//-------------------------------------------------------------------------------------------------------------------
//-- Stop --
	//
	TPL.FC_FirstStep(udiStepIndex, diStep);
	astStopTable[udiStepIndex].sTitle						:= 'Stop AllSubModules';
	astStopTable[udiStepIndex].udiModuleName				:= TPL.Gc_udiAllSubModules;
	astStopTable[udiStepIndex].diStep						:= diStep;
	astStopTable[udiStepIndex].diCMD						:= AXM.ET_Cmd.Stop;
	astStopTable[udiStepIndex].timTimeOut					:= T#0MS;
	astStopTable[udiStepIndex].xEndCMD						:= FALSE;
	
	TPL.FC_LastStep(udiStepIndex, diStep);
	astStopTable[udiStepIndex].sTitle						:= 'End';
	astStopTable[udiStepIndex].udiModuleName				:= 0;
	astStopTable[udiStepIndex].diStep						:= diStep;
	astStopTable[udiStepIndex].diCMD						:= 0;
	astStopTable[udiStepIndex].timTimeOut					:= T#0MS;
	astStopTable[udiStepIndex].xEndCMD						:= TRUE;
	
	TPL.FC_NextCmdTable(iq_udiTableIndex:= udiTableIndex);
	astListofCMDTables[udiTableIndex].sTitle				:= 'Stop';
	astListofCMDTables[udiTableIndex].diCMD					:= ET_Cmd.Stop;
	astListofCMDTables[udiTableIndex].udiNumberOfCmdSteps	:= udiStepIndex;

//-------------------------------------------------------------------------------------------------------------------
//-- Start --
	//
	TPL.FC_FirstStep(udiStepIndex, diStep);
	astStartTable[udiStepIndex].sTitle						:= 'Start AllSubModules';
	astStartTable[udiStepIndex].udiModuleName				:= TPL.Gc_udiAllSubModules;
	astStartTable[udiStepIndex].diStep						:= diStep;
	astStartTable[udiStepIndex].diCMD						:= AXM.ET_Cmd.Start;
	astStartTable[udiStepIndex].timTimeOut					:= T#0MS;
	astStartTable[udiStepIndex].xEndCMD						:= FALSE;
	
	TPL.FC_LastStep(udiStepIndex, diStep);
	astStartTable[udiStepIndex].sTitle						:= 'End';
	astStartTable[udiStepIndex].udiModuleName				:= 0;
	astStartTable[udiStepIndex].diStep						:= diStep;
	astStartTable[udiStepIndex].diCMD						:= 0;
	astStartTable[udiStepIndex].timTimeOut					:= T#0MS;
	astStartTable[udiStepIndex].xEndCMD						:= TRUE;
	
	TPL.FC_NextCmdTable(iq_udiTableIndex:= udiTableIndex);
	astListofCMDTables[udiTableIndex].sTitle				:= 'Start';
	astListofCMDTables[udiTableIndex].diCMD					:= ET_Cmd.Start;
	astListofCMDTables[udiTableIndex].udiNumberOfCmdSteps	:= udiStepIndex;
	
//-------------------------------------------------------------------------------------------------------------------
//-- Abort --
	//
	TPL.FC_FirstStep(udiStepIndex, diStep);
	astAbortTable[udiStepIndex].sTitle						:= 'Stop AllSubModules';
	astAbortTable[udiStepIndex].udiModuleName				:= TPL.Gc_udiAllSubModules;
	astAbortTable[udiStepIndex].diStep						:= diStep;
	astAbortTable[udiStepIndex].diCMD						:= AXM.ET_Cmd.Stop;
	astAbortTable[udiStepIndex].timTimeOut					:= T#0MS;
	astAbortTable[udiStepIndex].xEndCMD						:= FALSE;
	
	TPL.FC_LastStep(udiStepIndex, diStep);
	astAbortTable[udiStepIndex].sTitle						:= 	'End';
	astAbortTable[udiStepIndex].udiModuleName				:= 	0;
	astAbortTable[udiStepIndex].diStep						:= 	diStep;
	astAbortTable[udiStepIndex].diCMD						:= 	0;
	astAbortTable[udiStepIndex].timTimeOut					:=	T#0MS;
	astAbortTable[udiStepIndex].xEndCMD						:= TRUE;
	
	TPL.FC_NextCmdTable(iq_udiTableIndex:= udiTableIndex);
	astListofCMDTables[udiTableIndex].sTitle				:= 'Abort';
	astListofCMDTables[udiTableIndex].diCMD					:= ET_Cmd.Abort;
	astListofCMDTables[udiTableIndex].udiNumberOfCmdSteps	:= udiStepIndex;

//-------------------------------------------------------------------------------------------------------------------
//-- Hold --
	//
	TPL.FC_FirstStep(udiStepIndex, diStep);
	astHoldTable[udiStepIndex].sTitle						:= 'Hold AllSubModules';
	astHoldTable[udiStepIndex].udiModuleName				:= TPL.Gc_udiAllSubModules;
	astHoldTable[udiStepIndex].diStep						:= diStep;
	astHoldTable[udiStepIndex].diCMD						:= AXM.ET_Cmd.Hold;
	astHoldTable[udiStepIndex].timTimeOut					:= T#0MS;
	astHoldTable[udiStepIndex].xEndCMD						:= FALSE;
	
	TPL.FC_LastStep(udiStepIndex, diStep);
	astHoldTable[udiStepIndex].sTitle						:= 'End';
	astHoldTable[udiStepIndex].udiModuleName				:= 0;
	astHoldTable[udiStepIndex].diStep						:= diStep;
	astHoldTable[udiStepIndex].diCMD						:= 0;
	astHoldTable[udiStepIndex].timTimeOut					:= T#0MS;
	astHoldTable[udiStepIndex].xEndCMD						:= TRUE;
	
	TPL.FC_NextCmdTable(iq_udiTableIndex:= udiTableIndex);
	astListofCMDTables[udiTableIndex].sTitle				:= 'Hold';
	astListofCMDTables[udiTableIndex].diCMD					:= ET_Cmd.Hold;
	astListofCMDTables[udiTableIndex].udiNumberOfCmdSteps	:= udiStepIndex;

//-------------------------------------------------------------------------------------------------------------------
//-- Brake Release --
	//
	TPL.FC_FirstStep(udiStepIndex, diStep);
	astBrakeReleaseTable[udiStepIndex].sTitle				:= 'AxisEnable Off AllSubModules';
	astBrakeReleaseTable[udiStepIndex].udiModuleName		:= TPL.Gc_udiAllSubModules;
	astBrakeReleaseTable[udiStepIndex].diStep				:= diStep;
	astBrakeReleaseTable[udiStepIndex].diCMD				:= AXM.ET_Cmd.DriveEnableOff;
	astBrakeReleaseTable[udiStepIndex].timTimeOut			:= T#0MS;
	astBrakeReleaseTable[udiStepIndex].xEndCMD				:= FALSE;
	
	TPL.FC_NextStep(udiStepIndex, diStep);
	astBrakeReleaseTable[udiStepIndex].sTitle				:= 'BrakeRelease Mode AllSubModules';
	astBrakeReleaseTable[udiStepIndex].udiModuleName		:= TPL.Gc_udiAllSubModules;
	astBrakeReleaseTable[udiStepIndex].diStep				:= diStep;
	astBrakeReleaseTable[udiStepIndex].diCMD				:= AXM.ET_Cmd.BrakeRelease;
	astBrakeReleaseTable[udiStepIndex].timTimeOut			:= T#0MS;
	astBrakeReleaseTable[udiStepIndex].xEndCMD				:= FALSE;
	
	TPL.FC_NextStep(udiStepIndex, diStep);
	astBrakeReleaseTable[udiStepIndex].sTitle				:= 'Start AllSubModules';
	astBrakeReleaseTable[udiStepIndex].udiModuleName		:= TPL.Gc_udiAllSubModules;
	astBrakeReleaseTable[udiStepIndex].diStep				:= diStep;
	astBrakeReleaseTable[udiStepIndex].diCMD				:= AXM.ET_Cmd.Start;
	astBrakeReleaseTable[udiStepIndex].timTimeOut			:= T#0MS;
	astBrakeReleaseTable[udiStepIndex].xEndCMD				:= FALSE;
	
	TPL.FC_LastStep(udiStepIndex, diStep);
	astBrakeReleaseTable[udiStepIndex].sTitle				:= 'End';
	astBrakeReleaseTable[udiStepIndex].udiModuleName		:= 0;
	astBrakeReleaseTable[udiStepIndex].diStep				:= diStep;
	astBrakeReleaseTable[udiStepIndex].diCMD				:= 0;
	astBrakeReleaseTable[udiStepIndex].timTimeOut			:= T#0MS;
	astBrakeReleaseTable[udiStepIndex].xEndCMD				:= TRUE;
	
	TPL.FC_NextCmdTable(iq_udiTableIndex:= udiTableIndex);
	astListofCMDTables[udiTableIndex].sTitle				:= 'Brake Release';
	astListofCMDTables[udiTableIndex].diCMD					:= ET_Cmd.BrakeRelease;
	astListofCMDTables[udiTableIndex].udiNumberOfCmdSteps	:= udiStepIndex;
	//
//
			
// End of system generated code, could be modified for your application -)
END_ACTION

ACTION Init_SubModules:
(* System generated code, could be modified for your application *)

(*** Module Group declaration ***)

aaudiSubModuleGroups[c_udiBravoGroup1-TPL.Gc_udiGroupOffset,TPL.ET_Group.Member1] := 0;				(* There is no first element of the group c_diBravoGroup1 *)
aaudiSubModuleGroups[c_udiBravoGroup1-TPL.Gc_udiGroupOffset,TPL.ET_Group.Member2] := 0;				(* There is no second element of the group c_diBravoGroup1 *)

aaudiSubModuleGroups[c_udiBravoGroup2-TPL.Gc_udiGroupOffset,TPL.ET_Group.Member1] := c_udiSlave1;		(* The Slave1 is the first element of the group c_diBravoGroup2 *)
aaudiSubModuleGroups[c_udiBravoGroup2-TPL.Gc_udiGroupOffset,TPL.ET_Group.Member2] := c_udiSlave2;		(* The Slave2 is the second element of the group c_diBravoGroup2 *)

(* End of system generated code, could be modified for your application *)


(* System generated code, do not change without consulting 'Schneider Electric Automation GmbH' - otherwise you risk instability!!!*)
xInitSubModulesException := FALSE;

//-------------------------------------------------------------------------------------------------------------------
//-- Set IDs of SubModules *)	
//
	TPL.FC_SetSubModuleIds(	i_udiMainModuleID			:= iq_stStandardModuleItf.i_udiModuleId,
							i_pstSubModulesItf			:= ADR(astSubModuleInterface),
							i_udiNumberOfSubModules		:= c_udiNumberOfSubModules,
							q_etDiag					=> etDiag,
							q_etDiagExt					=> etDiagExtTPL);
	
	IF etDiag <> GD.ET_Diag.Ok AND NOT xInitSubModulesException THEN
		xInitSubModulesException := TRUE;
		
		stInitSubModulesException.sMsg := PDL.FC_MultiConcat(	i_sString1 := 'SetSubModuleIds - ', 
																i_sString2 := GD.FC_EtDiagToString(i_etDiag := etDiag), 
																i_sString3 := ' - ', 
																i_sString4 := TPL.FC_EtDiagExtToString(i_etDiagExt := etDiagExtTPL));
	END_IF	

//-------------------------------------------------------------------------------------------------------------------
//-- Set exception if any exception occurred *)
//
	fbExceptionHandler.SetException(i_xExceptionActive	:= xInitSubModulesException, 
									iq_stException		:= stInitSubModulesException, 
									iq_stExceptionList	:= iq_stExceptionList);
	
	xInitSuccessful := xInitSuccessful AND NOT xInitSubModulesException;
						
	etDiag := GD.ET_Diag.Ok;
(* End of system generated code, do not change without consulting 'Schneider Electric Automation GmbH' - otherwise you risk instability!!!*)
END_ACTION

ACTION ExceptionControl_Action:
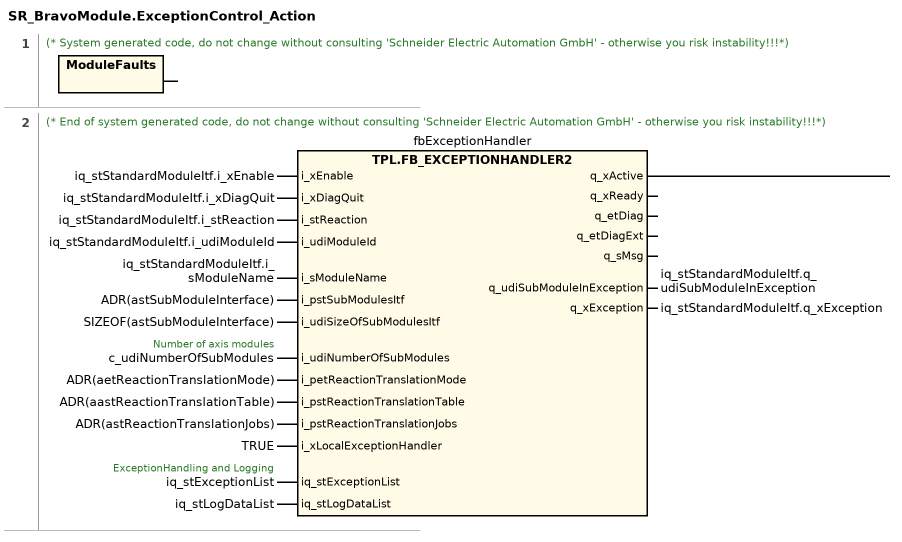
// NETWORK 1
// (* System generated code, do not change without consulting 'Schneider Electric Automation GmbH' - otherwise you risk instability!!!*)
ModuleFaults();

// NETWORK 2
// (* End of system generated code, do not change without consulting 'Schneider Electric Automation GmbH' - otherwise you risk instability!!!*)
//   fbExceptionHandler: ExceptionHandling related variables
//   c_udiNumberOfSubModules: Number of axis modules
//   iq_stExceptionList: ExceptionHandling and Logging
fbExceptionHandler(
    i_xEnable := iq_stStandardModuleItf.i_xEnable,
    i_xDiagQuit := iq_stStandardModuleItf.i_xDiagQuit,
    i_stReaction := iq_stStandardModuleItf.i_stReaction,
    i_udiModuleId := iq_stStandardModuleItf.i_udiModuleId,
    i_sModuleName := iq_stStandardModuleItf.i_sModuleName,
    i_pstSubModulesItf := ADR(astSubModuleInterface),
    i_udiSizeOfSubModulesItf := SIZEOF(astSubModuleInterface),
    i_udiNumberOfSubModules := c_udiNumberOfSubModules,
    i_petReactionTranslationMode := ADR(aetReactionTranslationMode),
    i_pstReactionTranslationTable := ADR(aastReactionTranslationTable),
    i_pstReactionTranslationJobs := ADR(astReactionTranslationJobs),
    i_xLocalExceptionHandler := TRUE,
    iq_stExceptionList := iq_stExceptionList,
    iq_stLogDataList := iq_stLogDataList,
    q_udiSubModuleInException => iq_stStandardModuleItf.q_udiSubModuleInException,
    q_xException => iq_stStandardModuleItf.q_xException); // TPL.FB_EXCEPTIONHANDLER2
END_ACTION

ACTION Init_Exceptions:
(* System generated code, could be modified for your application *)
stUpdateStructsException.etDiag												:= GD.ET_Diag.UnexpectedProgramBehavior;
stUpdateStructsException.udiDiagExt											:= ET_DiagExt.UpdateStructsException;
stUpdateStructsException.sDiagExt											:= FC_EtDiagExtToString(stUpdateStructsException.udiDiagExt);
stUpdateStructsException.sMsg												:= '';	(* Replaced on usage *)
stUpdateStructsException.udiModuleId										:= iq_stStandardModuleItf.i_udiModuleId;
stUpdateStructsException.sModuleName										:= iq_stStandardModuleItf.i_sModuleName;
stUpdateStructsException.stReaction.axReaction[TPL.ET_Reaction.AsyncStop]	:= TRUE;
stUpdateStructsException.etSource											:= TPL.ET_ExceptionSource.NodeModule;
stUpdateStructsException.timDelayTime										:= T#0MS;
stUpdateStructsException.wHmiAttributes										:= 0;
stUpdateStructsException.xAutoQuit											:= FALSE;

stInitReactionsException.etDiag												:= GD.ET_Diag.UnexpectedProgramBehavior;
stInitReactionsException.udiDiagExt											:= ET_DiagExt.InitReactionsException;
stInitReactionsException.sDiagExt											:= FC_EtDiagExtToString(stInitReactionsException.udiDiagExt);
stInitReactionsException.sMsg												:= '';	(* Replaced on usage *)
stInitReactionsException.udiModuleId										:= iq_stStandardModuleItf.i_udiModuleId;
stInitReactionsException.sModuleName										:= iq_stStandardModuleItf.i_sModuleName;
stInitReactionsException.stReaction.axReaction[TPL.ET_Reaction.AsyncStop]	:= TRUE;
stInitReactionsException.etSource											:= TPL.ET_ExceptionSource.NodeModule;
stInitReactionsException.timDelayTime										:= T#0MS;
stInitReactionsException.wHmiAttributes										:= 0;
stInitReactionsException.xAutoQuit											:= FALSE;

stInitSubModulesException.etDiag											:= GD.ET_Diag.UnexpectedProgramBehavior;
stInitSubModulesException.udiDiagExt										:= ET_DiagExt.InitSubModulesException;
stInitSubModulesException.sDiagExt											:= FC_EtDiagExtToString(stInitSubModulesException.udiDiagExt);
stInitSubModulesException.sMsg												:= '';	(* Replaced on usage *)
stInitSubModulesException.udiModuleId										:= iq_stStandardModuleItf.i_udiModuleId;
stInitSubModulesException.sModuleName										:= iq_stStandardModuleItf.i_sModuleName;
stInitSubModulesException.stReaction.axReaction[TPL.ET_Reaction.AsyncStop]	:= TRUE;
stInitSubModulesException.etSource											:= TPL.ET_ExceptionSource.NodeModule;
stInitSubModulesException.timDelayTime										:= T#0MS;
stInitSubModulesException.wHmiAttributes									:= 0;
stInitSubModulesException.xAutoQuit											:= FALSE;

stIsDriveVirtualException.etDiag											:= GD.ET_Diag.InputParameterInvalid;
stIsDriveVirtualException.udiDiagExt										:= ET_DiagExt.ifMulticarrierSegmentsInvalid ;
stIsDriveVirtualException.sDiagExt											:= FC_EtDiagExtToString(stIsDriveVirtualException.udiDiagExt);
stIsDriveVirtualException.sMsg												:= '';	(* Replaced on usage *)
stIsDriveVirtualException.udiModuleId										:= iq_stStandardModuleItf.i_udiModuleId;
stIsDriveVirtualException.sModuleName										:= iq_stStandardModuleItf.i_sModuleName;
stIsDriveVirtualException.stReaction.axReaction[TPL.ET_Reaction.AsyncStop]	:= TRUE;
stIsDriveVirtualException.etSource											:= TPL.ET_ExceptionSource.NodeModule;
stIsDriveVirtualException.timDelayTime										:= T#0MS;
stIsDriveVirtualException.wHmiAttributes									:= 0;
stIsDriveVirtualException.xAutoQuit											:= FALSE;

(*------------------------------------------------------------------------------------------*)
(* Init User Exceptions *)

	// TPL.ET_Reaction.AsyncStop
	// TPL.ET_Reaction.SyncStopEL
	// TPL.ET_Reaction.SyncStopEH
	// TPL.ET_Reaction.StopEndOfCycle
	// TPL.ET_Reaction.MainsContactorOff
	
(*------------------------------------------------------------------------------------------*)
stUserException1.etDiag													:= GD.ET_Diag.ExecutionAborted;
stUserException1.udiDiagExt												:= ET_DiagExtUser.Exception1FromEquipmentModule;
stUserException1.sDiagExt												:= FC_EtDiagExtUserToString(stUserException1.udiDiagExt);
stUserException1.sMsg													:= 'User Exception 1';
stUserException1.udiModuleId											:= iq_stStandardModuleItf.i_udiModuleId;
stUserException1.sModuleName											:= iq_stStandardModuleItf.i_sModuleName;
stUserException1.stReaction.axReaction[TPL.Gc_udiUserReactionOffset+2]	:= TRUE;
stUserException1.etSource												:= TPL.ET_ExceptionSource.User;
stUserException1.timDelayTime											:= T#0MS;
stUserException1.wHmiAttributes											:= 0;
stUserException1.xAutoQuit												:= FALSE;

stUserException2.etDiag													:= GD.ET_Diag.ExecutionAborted;
stUserException2.udiDiagExt												:= ET_DiagExtUser.Exception2FromEquipmentModule;
stUserException2.sDiagExt												:= FC_EtDiagExtUserToString(stUserException2.udiDiagExt);
stUserException2.sMsg													:= 'User Exception 2';
stUserException2.udiModuleId											:= iq_stStandardModuleItf.i_udiModuleId;
stUserException2.sModuleName											:= iq_stStandardModuleItf.i_sModuleName;
stUserException2.stReaction.axReaction[TPL.Gc_udiUserReactionOffset+2]	:= TRUE;
stUserException2.etSource												:= TPL.ET_ExceptionSource.User;
stUserException2.timDelayTime											:= T#0MS;
stUserException2.wHmiAttributes											:= 0;
stUserException2.xAutoQuit												:= FALSE;

(* End of system generated code, could be modified for your application *)
END_ACTION

ACTION Init_Reactions:
(* System generated code, only to be changed by experienced programmers *)
IF c_udiNumberOfSubModules < 1 THEN
	RETURN;
END_IF

(* Change of default reactions only on demand *)
(* Compare SR MainMachine Action Init_Reactions *)

xInitReactionsException := FALSE;

(*****************************************************************************************************************************************************)
(* Init ReactionTranslationMode *)

TPL.FC_InitReactionTranslationMode(	i_udiNumberOfSubModules			:= c_udiNumberOfSubModules,
									i_petReactionTranslationMode	:= ADR(aetReactionTranslationMode),
									q_etDiag						=> etDiag,
									q_etDiagExt						=> etDiagExtTPL);
							
IF etDiag <> GD.ET_Diag.Ok AND NOT xInitReactionsException THEN
	xInitReactionsException := TRUE;
	
	stInitReactionsException.sMsg := PDL.FC_MultiConcat(i_sString1 := 'InitReactionTranslationMode - ', 
														i_sString2 := GD.FC_EtDiagToString(i_etDiag := etDiag), 
														i_sString3 := ' - ', 
														i_sString4 := TPL.FC_EtDiagExtToString(i_etDiagExt := etDiagExtTPL));
END_IF	

(*****************************************************************************************************************************************************)
(* Init ReactionTranslationTable *)	

TPL.FC_InitReactionTranslationTable(i_udiNumberOfSubModules			:= c_udiNumberOfSubModules,
									i_pstReactionTranslationTable	:= ADR(aastReactionTranslationTable),
									q_etDiag						=> etDiag,
									q_etDiagExt						=> etDiagExtTPL);
									
IF etDiag <> GD.ET_Diag.Ok AND NOT xInitReactionsException THEN
	xInitReactionsException := TRUE;
	
	stInitReactionsException.sMsg := PDL.FC_MultiConcat(i_sString1 := 'InitReactionTranslationTable - ', 
														i_sString2 := GD.FC_EtDiagToString(i_etDiag := etDiag), 
														i_sString3 := ' - ', 
														i_sString4 := TPL.FC_EtDiagExtToString(i_etDiagExt := etDiagExtTPL));
END_IF		

(*****************************************************************************************************************************************************)
(* Init ReactionTranslationJobs *)	
								
TPL.FC_InitReactionTranslationJobs( i_udiNumberOfSubModules			:= c_udiNumberOfSubModules,
									i_pstReactionTranslationJobs	:= ADR(astReactionTranslationJobs),
									q_etDiag						=> etDiag,
									q_etDiagExt						=> etDiagExtTPL);
						
IF etDiag <> GD.ET_Diag.Ok AND NOT xInitReactionsException THEN
	xInitReactionsException := TRUE;
	
	stInitReactionsException.sMsg := PDL.FC_MultiConcat(i_sString1 := 'InitReactionTranslationJobs - ', 
														i_sString2 := GD.FC_EtDiagToString(i_etDiag := etDiag), 
														i_sString3 := ' - ', 
														i_sString4 := TPL.FC_EtDiagExtToString(i_etDiagExt := etDiagExtTPL));
END_IF		

(*****************************************************************************************************************************************************)
(* Set exception if any exception occurred *)

fbExceptionHandler.SetException(i_xExceptionActive	:= xInitReactionsException, 
								iq_stException		:= stInitReactionsException, 
								iq_stExceptionList	:= iq_stExceptionList);
					
xInitSuccessful := xInitSuccessful AND NOT xInitReactionsException;

etDiag := GD.ET_Diag.Ok;
(* End of system generated code, only to be changed by experienced programmers *)
END_ACTION

ACTION ModuleFaults:
(* System generated code, could be modified for your application *)
(* User Exception *)
fbExceptionHandler.SetException(	i_xExceptionActive	:= xModuleUserException1,
									iq_stException		:= stUserException1,
									iq_stExceptionList	:= iq_stExceptionList,
									q_etDiag			=> ,
									q_etDiagExt			=> ,
									q_sMsg				=> );

(* User Exception *)
fbExceptionHandler.SetException(	i_xExceptionActive	:= xModuleUserException2,
									iq_stException		:= stUserException2,
									iq_stExceptionList	:= iq_stExceptionList,
									q_etDiag			=> ,
									q_etDiagExt			=> ,
									q_sMsg				=> );

(* end of System generated code, could be modified for your application *)
END_ACTION

METHOD RegisterLoggerPoint
VAR_INPUT
	i_ifParent	: APL.IF_LoggerPoint;
	i_sName		: STRING[80];
END_VAR
VAR_OUTPUT
	q_etDiag	: GD.ET_Diag := GD.ET_Diag.Ok;
	q_etDiagExt	: ET_DiagExt := ET_DiagExt.Ok;
END_VAR
fbLoggerPoint.RegisterLoggerPoint(	i_ifParent	:= i_ifParent,
									i_sName		:= i_sName,
									i_sType		:= 'Node Module',
									i_sSource	:= 'Program',
									q_etDiag	=> ,
									q_etDiagExt	=> );
END_METHOD

ACTION InitModule_Action:
(* This step is used for initialisations after being enabled *)

(* System generated code, could be modified for your application *)
xInitSuccessful := TRUE;

Init_Exceptions();
(* End of system generated code, could be modified for your application *)

(* System generated code, do not change without consulting 'Schneider Electric Automation GmbH' - otherwise you risk instability!!!*)
iq_stStandardModuleItf.q_xActive		:= TRUE;
iq_stStandardModuleItf.q_xReady			:= FALSE;
iq_stStandardModuleItf.q_etDiag			:= GD.ET_Diag.Ok;
iq_stStandardModuleItf.q_udiDiagExt		:= ET_DiagExt.Initializing;
iq_stStandardModuleItf.q_sDiagExt		:= FC_EtDiagExtToString(ET_DiagExt.Initializing);
iq_stStandardModuleItf.q_sMsg			:= '';

Init_SubModules();
Init_CmdTables();
Init_Reactions();
UpdateStructs();
(* End of system generated code, do not change without consulting 'Schneider Electric Automation GmbH' - otherwise you risk instability!!!*)

(* System generated code, could be modified for your application *)
(*fbModuleController.RegisterLoggerPoint(	i_ifParent	:= fbLoggerPoint,
										i_sName		:= 'ModuleController',
										q_etDiag	=> ,
										q_etDiagExt	=> );
fbExceptionHandler.RegisterLoggerPoint(	i_ifParent	:= fbLoggerPoint,
										i_sName		:= 'ExceptionHandler',
										q_etDiag	=> ,
										q_etDiagExt	=> );*)
Init_Slave1();
Init_Slave2();
(* End of system generated code, could be modified for your application *)

(* Application specific code *)
(* ToDo: Add your application specific code here *)
;
(* End of application specific code *)
END_ACTION

ACTION Input_Action:
(* System generated code, do not change without consulting 'Schneider Electric Automation GmbH' - otherwise you risk instability!!!*)
UpdateStructs();
(* End of system generated code, do not change without consulting 'Schneider Electric Automation GmbH' - otherwise you risk instability!!!*)
END_ACTION

ACTION Logger_Action:
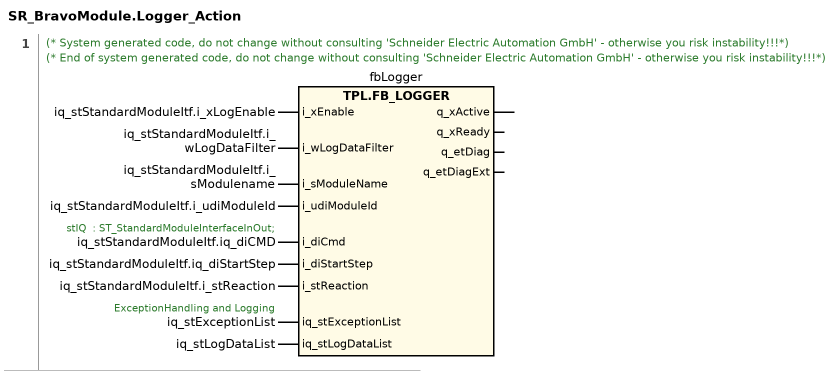
// NETWORK 1
// 					(* System generated code, do not change without consulting 'Schneider Electric Automation GmbH' - otherwise you risk instability!!!*)
// (* End of system generated code, do not change without consulting 'Schneider Electric Automation GmbH' - otherwise you risk instability!!!*)
//
//   fbLogger: Logging related variables
//   iq_stStandardModuleItf.iq_diCMD: stIQ : ST_StandardModuleInterfaceInOut;
//   iq_stExceptionList: ExceptionHandling and Logging
fbLogger(
    i_xEnable := iq_stStandardModuleItf.i_xLogEnable,
    i_wLogDataFilter := iq_stStandardModuleItf.i_wLogDataFilter,
    i_sModuleName := iq_stStandardModuleItf.i_sModulename,
    i_udiModuleId := iq_stStandardModuleItf.i_udiModuleId,
    i_diCmd := iq_stStandardModuleItf.iq_diCMD,
    i_diStartStep := iq_stStandardModuleItf.iq_diStartStep,
    i_stReaction := iq_stStandardModuleItf.i_stReaction,
    iq_stExceptionList := iq_stExceptionList,
    iq_stLogDataList := iq_stLogDataList); // TPL.FB_LOGGER
END_ACTION

ACTION Logic_active:
Check_RTB();
END_ACTION

ACTION Mode_Select:

END_ACTION

ACTION Output_Active:
(* System generated code, only to be changed by experienced programmers *)
IF iq_stStandardModuleItf.q_udiSubModuleInException <> 0 THEN
	iq_stStandardModuleItf.q_etDiag		:= GD.ET_Diag.Ok;
	iq_stStandardModuleItf.q_udiDiagExt	:= ET_DiagExt.SubModuleInException;
	iq_stStandardModuleItf.q_sDiagExt		:= FC_EtDiagExtToString(ET_DiagExt.SubModuleInException);
	iq_stStandardModuleItf.q_sMsg			:= '';
ELSE
	IF etDiagModuleController = GD.ET_Diag.Ok THEN
		iq_stStandardModuleItf.q_etDiag	:= etDiagModuleController;
		iq_stStandardModuleItf.q_sMsg		:= sMsgModuleController;
		
		CASE etDiagExtModuleController OF
			TPL.ET_DiagExt.DeactivatingSubModules : 
				iq_stStandardModuleItf.q_udiDiagExt	:= ET_DiagExt.DeactivatingSubModules;
				iq_stStandardModuleItf.q_sDiagExt		:= FC_EtDiagExtToString(ET_DiagExt.DeactivatingSubModules);
			TPL.ET_DiagExt.Disabled : 
				iq_stStandardModuleItf.q_udiDiagExt	:= ET_DiagExt.Disabled;
				iq_stStandardModuleItf.q_sDiagExt		:= FC_EtDiagExtToString(ET_DiagExt.Disabled);
			TPL.ET_DiagExt.ExecuteStep : 
				iq_stStandardModuleItf.q_udiDiagExt	:= ET_DiagExt.ExecuteStep;
				iq_stStandardModuleItf.q_sDiagExt		:= FC_EtDiagExtToString(ET_DiagExt.ExecuteStep);
			TPL.ET_DiagExt.Initializing : 
				iq_stStandardModuleItf.q_udiDiagExt	:= ET_DiagExt.Initializing;
				iq_stStandardModuleItf.q_sDiagExt		:= FC_EtDiagExtToString(ET_DiagExt.Initializing);
			TPL.ET_DiagExt.WaitAtNegativeStep : 
				iq_stStandardModuleItf.q_udiDiagExt	:= ET_DiagExt.WaitAtNegativeStep;
				iq_stStandardModuleItf.q_sDiagExt		:= FC_EtDiagExtToString(ET_DiagExt.WaitAtNegativeStep);
			TPL.ET_DiagExt.WaitCmdsDone : 
				iq_stStandardModuleItf.q_udiDiagExt	:= ET_DiagExt.WaitCmdsDone;
				iq_stStandardModuleItf.q_sDiagExt		:= FC_EtDiagExtToString(ET_DiagExt.WaitCmdsDone);
			TPL.ET_DiagExt.WaitForCmd : 
				iq_stStandardModuleItf.q_udiDiagExt	:= ET_DiagExt.WaitForCmd;
				iq_stStandardModuleItf.q_sDiagExt		:= FC_EtDiagExtToString(ET_DiagExt.WaitForCmd);
			ELSE
				iq_stStandardModuleItf.q_etDiag		:= GD. ET_Diag.UnexpectedProgramBehavior;
				iq_stStandardModuleItf.q_udiDiagExt	:= ET_DiagExt.UnknownStateModuleController;
				iq_stStandardModuleItf.q_sDiagExt		:= FC_EtDiagExtToString(ET_DiagExt.UnknownStateModuleController);
		END_CASE
	ELSE
		iq_stStandardModuleItf.q_etDiag		:= GD.ET_Diag.DiagActive;
		iq_stStandardModuleItf.q_udiDiagExt	:= ET_DiagExt.ModuleControllerException;
		iq_stStandardModuleItf.q_sDiagExt		:= FC_EtDiagExtToString(ET_DiagExt.ModuleControllerException);
		iq_stStandardModuleItf.q_sMsg			:= PDL.FC_MultiConcat(	i_sString1 := GD.FC_EtDiagToString(i_etDiag := etDiagModuleController), 
																			i_sString2 := ' - ',
																			i_sString3 := TPL.FC_EtDiagExtToString(etDiagExtModuleController), 
																			i_sString4 := '');
	END_IF
END_IF

(* End of system generated code, only to be changed by experienced programmers *)
END_ACTION

ACTION Start_Action:
(* This step is active until the machine is being enabled *)

(* System generated code, do not change without consulting 'Schneider Electric Automation GmbH' - otherwise you risk instability!!! *)
iq_stStandardModuleItf.q_xActive			:= FALSE;
iq_stStandardModuleItf.q_xReady			:= FALSE;

iq_stStandardModuleItf.q_etDiag			:= GD.ET_Diag.Ok;
iq_stStandardModuleItf.q_udiDiagExt		:= ET_DiagExt.Disabled;
iq_stStandardModuleItf.q_sDiagExt			:= FC_EtDiagExtToString(iq_stStandardModuleItf.q_udiDiagExt);
iq_stStandardModuleItf.q_sMsg				:= '';

iq_stStandardModuleItf.q_dwModuleType		:= TPL.ET_ModuleType.NodeModule;
iq_stStandardModuleItf.q_sModuleTypeName	:= 'NodeModule';
iq_stStandardModuleItf.q_udiModuleVersion	:= 1;	
(* End of system generated code, do not change without consulting 'Schneider Electric Automation GmbH' - otherwise you risk instability!!! *)

(* System generated code, to be changed by experienced programmers *)
IF iq_stStandardModuleItf.iq_diCMD <> 0 AND NOT iq_stStandardModuleItf.i_xEnable THEN
	iq_stStandardModuleItf.iq_diCMD := 0;
END_IF
(* End of system generated code, to be changed by experienced programmers *)

(* Application specific code *)
(* ToDo: Add your application specific code here *)
;
(* End of application specific code *)
END_ACTION

ACTION SubModules_Action:
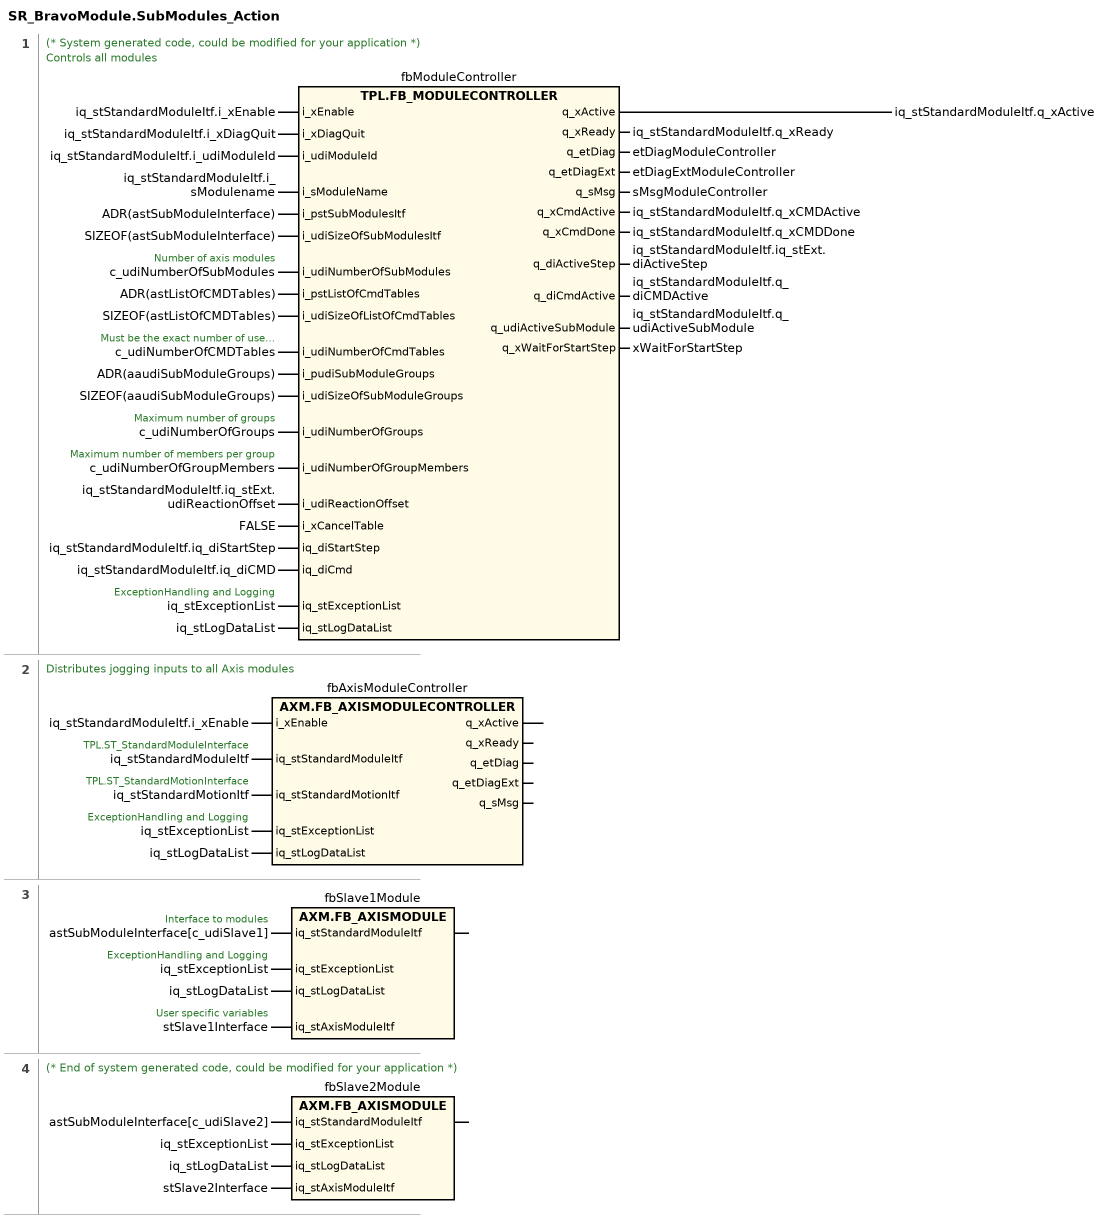
// NETWORK 1
// 					(* System generated code, could be modified for your application *)
// Controls all modules
//
//   fbModuleController: Modules related variables
//   c_udiNumberOfSubModules: Number of axis modules
//   c_udiNumberOfCMDTables: Must be the exact number of used CMDTables!
//   c_udiNumberOfGroups: Maximum number of groups
//   c_udiNumberOfGroupMembers: Maximum number of members per group
//   iq_stExceptionList: ExceptionHandling and Logging
fbModuleController(
    i_xEnable := iq_stStandardModuleItf.i_xEnable,
    i_xDiagQuit := iq_stStandardModuleItf.i_xDiagQuit,
    i_udiModuleId := iq_stStandardModuleItf.i_udiModuleId,
    i_sModuleName := iq_stStandardModuleItf.i_sModulename,
    i_pstSubModulesItf := ADR(astSubModuleInterface),
    i_udiSizeOfSubModulesItf := SIZEOF(astSubModuleInterface),
    i_udiNumberOfSubModules := c_udiNumberOfSubModules,
    i_pstListOfCmdTables := ADR(astListOfCMDTables),
    i_udiSizeOfListOfCmdTables := SIZEOF(astListOfCMDTables),
    i_udiNumberOfCmdTables := c_udiNumberOfCMDTables,
    i_pudiSubModuleGroups := ADR(aaudiSubModuleGroups),
    i_udiSizeOfSubModuleGroups := SIZEOF(aaudiSubModuleGroups),
    i_udiNumberOfGroups := c_udiNumberOfGroups,
    i_udiNumberOfGroupMembers := c_udiNumberOfGroupMembers,
    i_udiReactionOffset := iq_stStandardModuleItf.iq_stExt.udiReactionOffset,
    i_xCancelTable := FALSE,
    iq_diStartStep := iq_stStandardModuleItf.iq_diStartStep,
    iq_diCmd := iq_stStandardModuleItf.iq_diCMD,
    iq_stExceptionList := iq_stExceptionList,
    iq_stLogDataList := iq_stLogDataList,
    q_xReady => iq_stStandardModuleItf.q_xReady,
    q_etDiag => etDiagModuleController,
    q_etDiagExt => etDiagExtModuleController,
    q_sMsg => sMsgModuleController,
    q_xCmdActive => iq_stStandardModuleItf.q_xCMDActive,
    q_xCmdDone => iq_stStandardModuleItf.q_xCMDDone,
    q_diActiveStep => iq_stStandardModuleItf.iq_stExt.diActiveStep,
    q_diCmdActive => iq_stStandardModuleItf.q_diCMDActive,
    q_udiActiveSubModule => iq_stStandardModuleItf.q_udiActiveSubModule,
    q_xWaitForStartStep => xWaitForStartStep); // TPL.FB_MODULECONTROLLER
iq_stStandardModuleItf.q_xActive := fbModuleController.q_xActive;

// NETWORK 2
// Distributes jogging inputs to all Axis modules
//   iq_stStandardModuleItf: TPL.ST_StandardModuleInterface
//   iq_stStandardMotionItf: TPL.ST_StandardMotionInterface
//   iq_stExceptionList: ExceptionHandling and Logging
fbAxisModuleController(
    i_xEnable := iq_stStandardModuleItf.i_xEnable,
    iq_stStandardModuleItf := iq_stStandardModuleItf,
    iq_stStandardMotionItf := iq_stStandardMotionItf,
    iq_stExceptionList := iq_stExceptionList,
    iq_stLogDataList := iq_stLogDataList); // AXM.FB_AXISMODULECONTROLLER

// NETWORK 3
//   astSubModuleInterface[c_udiSlave1]: Interface to modules
//   iq_stExceptionList: ExceptionHandling and Logging
//   stSlave1Interface: User specific variables
fbSlave1Module(
    iq_stStandardModuleItf := astSubModuleInterface[c_udiSlave1],
    iq_stExceptionList := iq_stExceptionList,
    iq_stLogDataList := iq_stLogDataList,
    iq_stAxisModuleItf := stSlave1Interface); // AXM.FB_AXISMODULE

// NETWORK 4
// (* End of system generated code, could be modified for your application *)
fbSlave2Module(
    iq_stStandardModuleItf := astSubModuleInterface[c_udiSlave2],
    iq_stExceptionList := iq_stExceptionList,
    iq_stLogDataList := iq_stLogDataList,
    iq_stAxisModuleItf := stSlave2Interface); // AXM.FB_AXISMODULE
END_ACTION

ACTION UpdateStructs:
(* System generated code, do not change without consulting 'Schneider Electric Automation GmbH' - otherwise you risk instability!!!*)
fbDetectOnlineChange(	i_xEnable	:= TRUE, 
						i_xDetect	:= TRUE, 
						q_xActive	=> xDetectOnlineChangeActive, 
						q_xReady	=> xDetectOnlineChangeReady, 
						q_etDiag	=> etDetectOnlineChangeDiag, 
						q_etDiagExt	=> etDetectOnlineChangeDiagExt, 
						q_sMsg		=> sDetectOnlineChangeMsg, 
						q_xChange	=> );
						
IF(NOT fbDetectOnlineChange.q_xChange) THEN
	RETURN;
END_IF

iq_stStandardModuleItf.iq_stExt.udiNumberOfSubModules 		:= c_udiNumberOfSubModules;
iq_stStandardModuleItf.iq_stExt.dwSubModulesItf		 		:= ADR(astSubModuleInterface);
iq_stStandardModuleItf.iq_stExt.pdwSubModulesAddItf		 	:= ADR(adwSubModuleAddInterfaces);
iq_stStandardModuleItf.iq_stExt.pstListofCMDTables			:= ADR(astListOfCMDTables);
iq_stStandardModuleItf.iq_stExt.udiNumberOfCmdTables		:= c_udiNumberOfCMDTables;
(* End of system generated code, do not change without consulting 'Schneider Electric Automation GmbH' - otherwise you risk instability!!!*)

(* System generated code, could be modified for your application *)
xUpdateStructsException := FALSE;

//-------------------------------------------------------------------------------------------------------------------
//-- Update CmdTable - Prepare 
	//
	TPL.FC_UpdateCmdTableListElement(	i_pstListofCmdTables	:= ADR(astListOfCmdTables),
										i_udiNumberOfCmdTables	:= c_udiNumberOfCmdTables,
										i_diCmd					:= ET_Cmd.Prepare,
										i_pstCmdTable			:= ADR(astPrepareTable),
										q_etDiag				=> etDiag,
										q_etDiagExt				=> etDiagExtTPL);
										
	IF etDiag <> GD.ET_Diag.Ok AND NOT xUpdateStructsException THEN
		xUpdateStructsException := TRUE;
		
		stUpdateStructsException.sMsg := PDL.FC_MultiConcat(i_sString1 := 'Update CmdTable: Prepare - ', 
															i_sString2 := GD.FC_EtDiagToString(i_etDiag := etDiag), 
															i_sString3 := ' - ', 
															i_sString4 := TPL.FC_EtDiagExtToString(i_etDiagExt := etDiagExtTPL));
	END_IF										

//-------------------------------------------------------------------------------------------------------------------
//-- Update CmdTable - Auto 
	//
	TPL.FC_UpdateCmdTableListElement(	i_pstListofCmdTables	:= ADR(astListOfCmdTables),
										i_udiNumberOfCmdTables	:= c_udiNumberOfCmdTables,
										i_diCmd					:= ET_Cmd.Auto,
										i_pstCmdTable			:= ADR(astAutoTable),
										q_etDiag				=> etDiag,
										q_etDiagExt				=> etDiagExtTPL);
										
	IF etDiag <> GD.ET_Diag.Ok AND NOT xUpdateStructsException THEN
		xUpdateStructsException := TRUE;
		
		stUpdateStructsException.sMsg := PDL.FC_MultiConcat(i_sString1 := 'Update CmdTable: Auto - ', 
															i_sString2 := GD.FC_EtDiagToString(i_etDiag := etDiag), 
															i_sString3 := ' - ', 
															i_sString4 := TPL.FC_EtDiagExtToString(i_etDiagExt := etDiagExtTPL));
	END_IF		

//-------------------------------------------------------------------------------------------------------------------
//-- Update CmdTable - Manual 
	//
	TPL.FC_UpdateCmdTableListElement(	i_pstListofCMDTables	:= ADR(astListofCMDTables),
										i_udiNumberOfCMDTables	:= c_udiNumberOfCMDTables,
										i_diCMD					:= ET_Cmd.Manual,
										i_pstCMDTable			:= ADR(astManualTable),
										q_etDiag				=> etDiag,
										q_etDiagExt				=> etDiagExtTPL);
										
	IF etDiag <> GD.ET_Diag.Ok AND NOT xUpdateStructsException THEN
		xUpdateStructsException := TRUE;
		
		stUpdateStructsException.sMsg := PDL.FC_MultiConcat(i_sString1 := 'Update CmdTable: Manual - ', 
															i_sString2 := GD.FC_EtDiagToString(i_etDiag := etDiag), 
															i_sString3 := ' - ', 
															i_sString4 := TPL.FC_EtDiagExtToString(i_etDiagExt := etDiagExtTPL));
	END_IF		

//-------------------------------------------------------------------------------------------------------------------
//-- Update CmdTable - Stop 
	//
	TPL.FC_UpdateCmdTableListElement(	i_pstListofCMDTables	:= ADR(astListofCMDTables),
										i_udiNumberOfCMDTables	:= c_udiNumberOfCMDTables,
										i_diCMD					:= ET_Cmd.Stop,
										i_pstCMDTable			:= ADR(astStopTable),
										q_etDiag				=> etDiag,
										q_etDiagExt				=> etDiagExtTPL);
										
	IF etDiag <> GD.ET_Diag.Ok AND NOT xUpdateStructsException THEN
		xUpdateStructsException := TRUE;
		
		stUpdateStructsException.sMsg := PDL.FC_MultiConcat(i_sString1 := 'Update CmdTable: Stop - ', 
															i_sString2 := GD.FC_EtDiagToString(i_etDiag := etDiag), 
															i_sString3 := ' - ', 
															i_sString4 := TPL.FC_EtDiagExtToString(i_etDiagExt := etDiagExtTPL));
	END_IF		

//-------------------------------------------------------------------------------------------------------------------
//-- Update CmdTable - Start 
	//
	TPL.FC_UpdateCmdTableListElement(	i_pstListofCMDTables	:= ADR(astListofCMDTables),
										i_udiNumberOfCmdTables	:= c_udiNumberOfCMDTables,
										i_diCMD					:= ET_Cmd.Start,
										i_pstCMDTable			:= ADR(astStartTable),
										q_etDiag				=> etDiag,
										q_etDiagExt				=> etDiagExtTPL);
										
	IF etDiag <> GD.ET_Diag.Ok AND NOT xUpdateStructsException THEN
		xUpdateStructsException := TRUE;
		
		stUpdateStructsException.sMsg := PDL.FC_MultiConcat(i_sString1 := 'Update CmdTable: Start - ', 
															i_sString2 := GD.FC_EtDiagToString(i_etDiag := etDiag), 
															i_sString3 := ' - ', 
															i_sString4 := TPL.FC_EtDiagExtToString(i_etDiagExt := etDiagExtTPL));
	END_IF		

//-------------------------------------------------------------------------------------------------------------------
//-- Update CmdTable - Abort 
	//
	TPL.FC_UpdateCmdTableListElement(	i_pstListofCMDTables	:= ADR(astListofCMDTables),
										i_udiNumberOfCmdTables	:= c_udiNumberOfCmdTables,
										i_diCMD					:= ET_Cmd.Abort,
										i_pstCMDTable			:= ADR(astAbortTable),
										q_etDiag				=> etDiag,
										q_etDiagExt				=> etDiagExtTPL);
										
	IF etDiag <> GD.ET_Diag.Ok AND NOT xUpdateStructsException THEN
		xUpdateStructsException := TRUE;
		
		stUpdateStructsException.sMsg := PDL.FC_MultiConcat(i_sString1 := 'Update CmdTable: Abort - ', 
															i_sString2 := GD.FC_EtDiagToString(i_etDiag := etDiag), 
															i_sString3 := ' - ', 
															i_sString4 := TPL.FC_EtDiagExtToString(i_etDiagExt := etDiagExtTPL));
	END_IF		

//-------------------------------------------------------------------------------------------------------------------
//-- Update CmdTable - Hold 
	//
	TPL.FC_UpdateCmdTableListElement(	i_pstListofCMDTables	:= ADR(astListofCMDTables),
										i_udiNumberOfCmdTables	:= c_udiNumberOfCmdTables,
										i_diCMD					:= ET_Cmd.Hold,
										i_pstCMDTable			:= ADR(astHoldTable),
										q_etDiag				=> etDiag,
										q_etDiagExt				=> etDiagExtTPL);
										
	IF etDiag <> GD.ET_Diag.Ok AND NOT xUpdateStructsException THEN
		xUpdateStructsException := TRUE;
		
		stUpdateStructsException.sMsg := PDL.FC_MultiConcat(i_sString1 := 'Update CmdTable: Hold - ', 
															i_sString2 := GD.FC_EtDiagToString(i_etDiag := etDiag), 
															i_sString3 := ' - ', 
															i_sString4 := TPL.FC_EtDiagExtToString(i_etDiagExt := etDiagExtTPL));
	END_IF		

//-------------------------------------------------------------------------------------------------------------------
//-- Update CmdTable - BrakeRelease 
	//
	TPL.FC_UpdateCmdTableListElement(	i_pstListofCMDTables	:= ADR(astListofCMDTables),
										i_udiNumberOfCMDTables	:= c_udiNumberOfCMDTables,
										i_diCMD					:= ET_Cmd.BrakeRelease,
										i_pstCMDTable			:= ADR(astBrakeReleaseTable),
										q_etDiag				=> etDiag,
										q_etDiagExt				=> etDiagExtTPL);
										
	IF etDiag <> GD.ET_Diag.Ok AND NOT xUpdateStructsException THEN
		xUpdateStructsException := TRUE;
		
		stUpdateStructsException.sMsg := PDL.FC_MultiConcat(i_sString1 := 'Update CmdTable: BrakeRelease - ', 
															i_sString2 := GD.FC_EtDiagToString(i_etDiag := etDiag), 
															i_sString3 := ' - ', 
															i_sString4 := TPL.FC_EtDiagExtToString(i_etDiagExt := etDiagExtTPL));
	END_IF		
									
				
//-------------------------------------------------------------------------------------------------------------------
//-- Update AddInterface - Slave1 
	//
	AXM.FC_UpdateAddInterfaceStruct(	i_pdwSubModuleAddInterfaces	:= ADR(adwSubModuleAddInterfaces),
										i_udiSubModuleConstant		:= c_udiSlave1,
										iq_stAxisModuleItf			:= stSlave1Interface,
										q_etDiag					=> etDiag,
										q_etDiagExt					=> etDiagExtAXM);
										
	IF etDiag <> GD.ET_Diag.Ok AND NOT xUpdateStructsException THEN
		xUpdateStructsException := TRUE;
		
		stUpdateStructsException.sMsg := PDL.FC_MultiConcat(i_sString1 := 'Update AddInterface: Slave1 - ', 
															i_sString2 := GD.FC_EtDiagToString(i_etDiag := etDiag), 
															i_sString3 := ' - ', 
															i_sString4 := AXM.FC_EtDiagExtToString(i_etDiagExt := etDiagExtAXM));
	END_IF		

//-------------------------------------------------------------------------------------------------------------------
//-- Update AddInterface - Slave2
	//
	AXM.FC_UpdateAddInterfaceStruct(	i_pdwSubModuleAddInterfaces	:= ADR(adwSubModuleAddInterfaces),
										i_udiSubModuleConstant		:= c_udiSlave2,
										iq_stAxisModuleItf			:= stSlave2Interface,
										q_etDiag					=> etDiag,
										q_etDiagExt					=> etDiagExtAXM);
										
	IF etDiag <> GD.ET_Diag.Ok AND NOT xUpdateStructsException THEN
		xUpdateStructsException := TRUE;
		
		stUpdateStructsException.sMsg := PDL.FC_MultiConcat(i_sString1 := 'Update AddInterface: Slave2 - ', 
															i_sString2 := GD.FC_EtDiagToString(i_etDiag := etDiag), 
															i_sString3 := ' - ', 
															i_sString4 := AXM.FC_EtDiagExtToString(i_etDiagExt := etDiagExtAXM));
	END_IF		

//-------------------------------------------------------------------------------------------------------------------
//-- Update ILS Data 
	//
	// stSlave1Interface.stEndless.pstIlsData	:= ADR(G_stIlsData);
	// stSlave1Interface.stMultiCam.pstIlsData	:= ADR(G_stIlsData);
	
	// stSlave2Interface.stEndless.pstIlsData	:= ADR(G_stIlsData);
	// stSlave2Interface.stMultiCam.pstIlsData	:= ADR(G_stIlsData);

//-------------------------------------------------------------------------------------------------------------------
//-- Set exception if any exception occurred *)
	//
	fbExceptionHandler.SetException(i_xExceptionActive	:= xUpdateStructsException, 
									iq_stException		:= stUpdateStructsException, 
									iq_stExceptionList	:= iq_stExceptionList);
									
	xInitSuccessful := xInitSuccessful AND NOT xUpdateStructsException;
	
	etDiag := GD.ET_Diag.Ok;
(* End of system generated code, could be modified for your application *)
END_ACTION

END_PROGRAM

// LMC_PacDrive/Application/TemplateFullProgrammingFramework/EquipmentModules/MulticarrierModule/SR_MulticarrierModule
PROGRAM SR_MulticarrierModule

VAR CONSTANT
	(* Standard related constants *)
		c_udiNumberOfGroups				: UDINT := 1;			(* Maximum number of groups *)
		c_udiNumberOfGroupMembers		: UDINT := 10;			(* Maximum number of members per group *)
	
		c_udiNumberOfCmdTables			: UDINT := 9;			(* Must be the exact number of used CMDTables! *)
		c_udiNumberOfCmdSteps			: UDINT := 16;			(* Make sure that the number of commands/ Steps  that each table
																	   contains does not exceed the c_diNumberOfCMDSteps variable.*)
	
	(* Definition group of modules *)
		c_udiMultiCarrierGroup1			: UDINT := 2001;		(* Name of module group  1 *)
	
	(* System generated code, could be modified for your application *)
		c_udiNumberOfSubModules			: UDINT := 1;			(* Number of axis modules *)
		c_udiMultiCarrierTrack			: UDINT := 1;
	(* End of system generated code, could be modified for your application *)
END_VAR

VAR_INPUT
	(* Master of MultiCarrierModule *)
		i_ifMaster						: SystemConfigurationItf.IF_Master;
END_VAR

VAR_IN_OUT
	(* TPL.ST_StandardModuleInterface *)	
		iq_stStandardModuleItf			: TPL.ST_StandardModuleInterface;
		
	(* TPL.ST_StandardMotionInterface *)		
		iq_stStandardMotionItf			: TPL.ST_StandardMotionInterface;
		
	(* ExceptionHandling and Logging *)	
		iq_stExceptionList				: TPL.ST_ExceptionList;
		iq_stLogDataList				: TPL.ST_LogDataList;
		iq_stMulticarrierModule			: ST_MulticarrierModule;
END_VAR

//--- user variables:
VAR

	xSetStationTriggerViaTimer	: BOOL;
	
	//-- Station1 -------------------------------------------------
	fbStation1						: FB_Station1;
	stStation1						: ST_StationParameter;
END_VAR

//--- fbMulticarrier 
VAR
//-- ErrorHandling ---------------------------------
	sEtResult						: STRING(255);
	udiEtResult						: UDINT;
	etResultSource					: ET_ResultSource;
	xErrorStored					: BOOL;
	etResultMCR						: MCR.ET_Result;
	etResultMCRS					: MCRS.ET_Result;
	sResultMsgMCR					: STRING(255);
	sResultMsg1						: STRING(80);
	sResultMsg2						: STRING(80);
	sResultMsg3						: STRING(80);
	xSetException					: BOOL;
	udiLoop							: UDINT;
	xErrorActive					: BOOL;
	xHomingWasSuccessful			: BOOL;
	uiSetOpModeVis					: UINT;
	
//--- Check RTB ---------------------------------
	diStateRTB						: DINT := 0;
	xRTBFailureFlag					: BOOL;
	udiCount						: UDINT;
	xModulesActive					: BOOL;
	xModulesNotActive				: BOOL;	

//--- Control Module ---------------------------------       		
	iStateOpMode					: INT:= 0;	
	fbRTrigCMDActive				: R_TRIG;
	fbRTrigError					: R_TRIG;
	etLastCmd						: ET_CMD;
	
//--- Init_Multicarrier ---------------------------------
	lrMaxDecelerationEmergency			: LREAL := 100_000.0;
	lrMaxAbsJerkEmergency				: LREAL := 1_000_000.0;
	lrRefMinGapToCarrierInFront			: LREAL := 15;
	lrRefMinGapToCarrierBehind			: LREAL := 15;

//--- fbMultiCarrier ---------------------------------------------------	
	ifMulticarrier						: MCR.IF_Multicarrier;
	fbMulticarrier						: MCR.FB_Multicarrier;
	xEnableFbMulticarrier				: BOOL;
	xStartFbMulticarrier				: BOOL;
	etResultFbMulticarrier				: MCR.ET_Result;
	sResultMsgFbMulticarrier			: STRING(255);
	
//--- fbCrashPrevention ---------------------------------------------------	
	fbCrashPrevention					: MCR.FB_CrashPrevention;
	xEnableFbCrashPrevention			: BOOL := FALSE;
	xStartFbCrashPrevention				: BOOL;
	xActiveFbCrashPrevention			: BOOL;
	xReadyFbCrashPrevention				: BOOL; 
	xErrorFbCrashPrevention				: BOOL; 
	etResultFbCrashPrevention			: MCR.ET_Result; 
	sResultMsgFbCrashPrevention			: string(255); 
	stFeedbackFbCrashPrevention			: MCR.ST_CrashPreventionFeedback;
	xErrorFbCrashPreventionStored		: BOOL;
	etResultFbCrashPreventionStored		: MCR.ET_Result;
	sResultMsgFbCrashPreventionStored	: STRING(255);
	stCrashPreventionParameterLocal		: MCR.ST_CrashPreventionParameter;
	
//--- Homing -----------------------
	audiOrderOfCarrier 					: ARRAY [1..MCR.GPl.Gc_udiMaxNumberOfCarriers] OF UDINT;
	udiNumberOfCarrier					: UDINT;

//--- Jogging -----------------------
	xSetCarrierForJoggingFromVis		: BOOL;
	udiJoggingCarrierNr					: UDINT;
	xSetJogAllCarrier					: BOOL;
	xSetJogSingleCarrier				: BOOL;
	xJogAllCarrier						: BOOL;
	iAxisSelect							: INT;
	xJogSingleCarrier					: BOOL := TRUE;
	xJogForw							: BOOL;
	xJogBack							: BOOL;
	xJogCarrierSelectEnableFlag			: BOOL;
	iJogMode							: INT;
	lrJogVelocity						: LREAL := 100;
	lrJogVelocityOld					: LREAL := 0;
	lrJogMinDistanceBetweenCarrier  	: LREAL := 100;
	lrJogMinDistanceBetweenCarrierOld	: LREAL := 0;
	alrStoredMinGapInFront				: ARRAY [1..MCR.GPL.Gc_udiMaxNumberOfCarriers] OF LREAL;
	alrStoredMinGapBehind				: ARRAY [1..MCR.GPL.Gc_udiMaxNumberOfCarriers] OF LREAL;

//--- ControlEnable ------------------	
	iStateControlEnable					: INT;
	xControlEnable						: BOOL;
	udiIndex							: UDINT;
	xEnableTrackSuccessful				: BOOL;
	diTimerStopOpmode					: DINT;
	diWaitTimeSetCarrierEnableFalse		: DINT := 1000; //[ms]
	xCheckTimeOutControlEnable			: BOOL;
	fbTonTimeOutControlEnable			: Standard.TON;
	timTimeoutControlEnable				: TIME := T#5000MS;
	
//--- Diagnostics ------------------
	etLogLevelMcr						: APL.ET_LogLevel := APL.ET_LogLevel.UserAction;
	etLogLevelMcrOld					: APL.ET_LogLevel := APL.ET_LogLevel.UserAction;
	xSetForAllAplMsg					: BOOL;
	xReSetForAllAplMsg					: BOOL;
	xSetSingleAplMsg					: BOOL;
	xAplMsgStartPosAndEndPos			: BOOL;
	lrAplStartTrackPos					: LREAL;
	lrAplEndTrackPos					: LREAL;
	udiDeltaBottomY						: UDINT := 1000;
	iTopTraceEntryVis					: INT;
	
	//--- FB_TrackCalibration
	fbTrackCalibration			: MCR.FB_TrackCalibration;
	xEnableFbTrackCalibration	: BOOL;
	xStartFbTrackCalibration	: BOOL;
	xActiveFbTrackCalibration	: BOOL;
	xReadyFbTrackCalibration	: BOOL;
	xErrorFbTrackCalibration	: BOOL;
	etResultFbTrackCalibration	: MCR.ET_Result;
	sResultMsgFbTrackCalibration: STRING(255);
	xStartCalibration			: BOOL;
	xStartMeasurement			: BOOL;
	xResetTrackCalibration		: BOOL;
	udiActiveJobs				: UDINT;
	udiCreatedTasks				: UDINT;
	udiPendingJobs				: UDINT;
	xInitDone					: BOOL;;
	etModeTrackCalibration		: MCR.ET_ModeTrackCalibration := MCR.ET_ModeTrackCalibration.Forward;
	
//--- IGOR: Delete Start
	iStateTrackPowerCycle		: DINT;
	xStartTrackPowerCycle		: BOOL;
	xActiveTrackPowerCycle		: BOOL;
	xFinishedTrackPowerCycle	: BOOL;
	diTimerTrackPowerCylcle		: DINT;
	diWaitTimeTrackDisable		: DINT := 2000;
	diWaitTimeTrackEnable		: DINT := 20000;		
	
	xTestStartDebugCalculationClockwise	: BOOL;
	alrHighestPositionJump		: ARRAY[1..MCR.GPL.Gc_udiMaxNumberOfSegments] OF LREAL := [0.267,0.318,0.411,0.5,0.086,0.19,0.101,0.045,0.237,0.098,0.213,0.282,0.076,0.444];//[0,0,0,0,0,1,0,0,0,0,0,0,0,0];
//--- IGOR: Delete End	

	
//--- Trace-------------------------
	etTraceSource						: ET_TraceSource;
	fbDummyFeedback						: MCR.FB_DummyCarrierFeedback;
	aifTraceObject						: ARRAY[1..5] OF MCR.IF_CarrierFeedback := [5(fbDummyFeedback)];
	udiTraceObject1						: UDINT := 1;
	udiTraceObject2						: UDINT := 2;
	udiTraceObject3						: UDINT := 3;
	udiTraceObject4						: UDINT := 4;
	udiTraceObject5						: UDINT := 5;
	aifTraceCarrierMovementData			: ARRAY[1..5] OF SystemUserFunctionsItf.IF_MovementData;
	xSetNewTraceObjects					: BOOL;
	udiNumberOfCarrierInTrace			: UDINT := 5;
	xReStartOneByOneCount				: BOOL;
	xOneByOne							: BOOL;
	udiSingleCarrierNr					: UDINT;
	lrTraceStartTrackPos				: LREAL;
	lrTraceEndTrackPos					: LREAL;

//--- Vis -------------------------
	aifVisFeedback						: ARRAY[1..150] OF MCR.IF_CarrierFeedback := [150(fbDummyFeedback)];
	udiVisLoop							: UDINT;
	uiAdditionalVisTabs					: UINT;
	fbErrorVisTabTrig					: Standard.R_TRIG;
	fbResetErrorVisTabTrig				: Standard.F_TRIG;
	etVisPosColumn1						: ET_VisPosGapDist := ET_VisPosGapDist.RefTrackPosition;
	etVisPosColumn2						: ET_VisPosGapDist := ET_VisPosGapDist.GapToCarrierInFront;
	etVisPosColumn3						: ET_VisPosGapDist := ET_VisPosGapDist.GapToCarrierBehind;
	
//--- TestStations ------------------------------------
	xStartTest							: BOOL;
	xStopTest							: BOOL;

//--- Template variables ---------------------------------
	xInitSuccessful : BOOL := FALSE;
		
(* Standard related variables *)
	astSubModuleInterface			: ARRAY[1..c_udiNumberOfSubModules] OF TPL.ST_StandardModuleInterface;		(* Interface to modules *)
	aaudiSubModuleGroups			: ARRAY[1..c_udiNumberOfGroups,1..c_udiNumberOfGroupMembers] OF UDINT;
	adwSubModuleAddInterfaces		: ARRAY[1..c_udiNumberOfSubModules] OF DWORD;
	
(* Modules related variables *)
	fbModuleController				: TPL.FB_ModuleController;
	etDiagModuleController			: GD.ET_Diag;
	etDiagExtModuleController		: TPL.ET_DiagExt;
	sMsgModuleController			: STRING[80];
	xWaitForStartStep				: BOOL;
	astListOfCmdTables				: ARRAY [1..c_udiNumberOfCmdTables] OF TPL.ST_CmdTable;
	udiTableIndex					: UDINT;
	udiStepIndex					: UDINT;
	diStep							: DINT;

	astPrepareTable					: ARRAY [1..c_udiNumberOfCmdSteps] OF TPL.ST_Cmd;		(* Relating  Cmd table *)
	astAutoTable					: ARRAY [1..c_udiNumberOfCmdSteps] OF TPL.ST_Cmd;		(* Relating  Cmd table *)
	astManualTable					: ARRAY [1..c_udiNumberOfCmdSteps] OF TPL.ST_Cmd;		(* Relating  Cmd table *)
	astHoldTable					: ARRAY [1..c_udiNumberOfCmdSteps] OF TPL.ST_Cmd;		(* Relating  Cmd table *)
	astStartTable					: ARRAY [1..c_udiNumberOfCmdSteps] OF TPL.ST_Cmd;		(* Relating  Cmd table *)
	astStopTable					: ARRAY [1..c_udiNumberOfCmdSteps] OF TPL.ST_Cmd;		(* Relating  Cmd table *)
	astAbortTable					: ARRAY [1..c_udiNumberOfCmdSteps] OF TPL.ST_Cmd;		(* Relating  Cmd table *)
	astTestMulticarrierTable	: ARRAY [1..c_udiNumberOfCmdSteps] OF TPL.ST_Cmd; (* Relating  Cmd table *)
	astTrackCalibrationTable		: ARRAY [1..c_udiNumberOfCmdSteps] OF TPL.ST_Cmd; 		(* Relating  Cmd table *)

(* ExceptionHandling related variables *)
	fbExceptionHandler				: TPL.FB_ExceptionHandler2;

	aetReactionTranslationMode		: ARRAY[1..c_udiNumberOfSubModules] OF TPL.ET_ReactionTranslationMode;
	aastReactionTranslationTable	: ARRAY[1..c_udiNumberOfSubModules,1..TPL.Gc_udiMaxNumberOfReactions] OF TPL.ST_Reaction;
	astReactionTranslationJobs		: ARRAY[1..c_udiNumberOfSubModules] OF TPL.ST_ReactionTranslationJobs;
	
(* Exception declaration *)

	stException						: TPL.ST_Exception;
	stHardwareException				: TPL.ST_Exception;
	
	stUpdateStructsException		: TPL.ST_Exception;
	xUpdateStructsException			: BOOL;
	
	stInitReactionsException		: TPL.ST_Exception;
	xInitReactionsException			: BOOL;
	
	stInitSubModulesException		: TPL.ST_Exception;
	xInitSubModulesException		: BOOL;
	
(* Logging related variables *)
	fbLogger						: TPL.FB_Logger;
	fbLoggerPoint					: APL.FB_LoggerPoint;

(* OnlineChange related variables *)
	fbDetectOnlineChange			: TPL.FB_DetectOnlineChange;
	xDetectOnlineChangeActive		: BOOL; 
	xDetectOnlineChangeReady		: BOOL; 
	etDetectOnlineChangeDiag		: GD.ET_Diag;
	etDetectOnlineChangeDiagExt		: TPL.ET_DiagExt; 
	sDetectOnlineChangeMsg			: STRING[80];
	
(* POU-Feedback related variables *)	
	etDiag			: GD.ET_Diag;
	etDiagExtTPL	: TPL.ET_DiagExt;
	
	//--- Hardwarefaults
	stDiagSource				: SystemConfiguration.ST_LogicalAddress;
	sInstanceName				: STRING[80];
	diDiagClass					: DINT;
	diDiagCode					: DINT;
	diDiagCode_old				: DINT;
	sDiagMsg					: STRING[40];
	sDiagMsgExt					: STRING[15];
	ifDiagnosis					: SystemConfigurationItf.IF_Diagnosis;
	xSuccess					: BOOL;


END_VAR

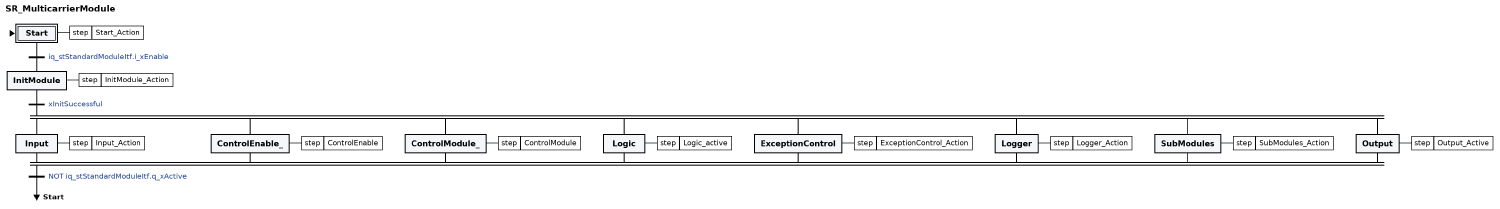
INITIAL_STEP Start:
    Start_Action(N);  // step action
END_STEP
TRANSITION FROM Start TO InitModule
    := iq_stStandardModuleItf.i_xEnable;
END_TRANSITION
STEP InitModule:
    InitModule_Action(N);  // step action
END_STEP
TRANSITION FROM InitModule TO (Input, ControlEnable_, ControlModule_, Logic, ExceptionControl, Logger, SubModules, Output)
    := xInitSuccessful;
END_TRANSITION
STEP Input:
    Input_Action(N);  // step action
END_STEP
STEP ControlEnable_:
    ControlEnable(N);  // step action
END_STEP
STEP ControlModule_:
    ControlModule(N);  // step action
END_STEP
STEP Logic:
    Logic_active(N);  // step action
END_STEP
STEP ExceptionControl:
    ExceptionControl_Action(N);  // step action
END_STEP
STEP Logger:
    Logger_Action(N);  // step action
END_STEP
STEP SubModules:
    SubModules_Action(N);  // step action
END_STEP
STEP Output:
    Output_Active(N);  // step action
END_STEP
TRANSITION FROM (Input, ControlEnable_, ControlModule_, Logic, ExceptionControl, Logger, SubModules, Output) TO Start
    := NOT iq_stStandardModuleItf.q_xActive;
END_TRANSITION

ACTION Init_CmdTables:
(* System generated code, could be modified for your application *)

//-------------------------------------------------------------------------------------------------------------------
//-- Prepare  --
	//
	TPL.FC_FirstStep(udiStepIndex, diStep);
	astPrepareTable[udiStepIndex].sTitle					:= 'Prepare MultiCarrier';
	astPrepareTable[udiStepIndex].udiModuleName				:= c_udiMultiCarrierTrack;
	astPrepareTable[udiStepIndex].diStep					:= -diStep;
	astPrepareTable[udiStepIndex].diCMD						:= 0;
	astPrepareTable[udiStepIndex].timTimeOut				:= T#0MS;
	astPrepareTable[udiStepIndex].xEndCMD					:= FALSE;
	
	TPL.FC_LastStep(udiStepIndex, diStep); 
	astPrepareTable[udiStepIndex].sTitle					:= 'End';
	astPrepareTable[udiStepIndex].udiModuleName				:= 0;
	astPrepareTable[udiStepIndex].diStep					:= diStep;
	astPrepareTable[udiStepIndex].diCMD						:= 0;
	astPrepareTable[udiStepIndex].timTimeOut				:= T#0MS;
	astPrepareTable[udiStepIndex].xEndCMD					:= TRUE;
	
	TPL.FC_FirstCmdTable(iq_udiTableIndex:= udiTableIndex);
	astListofCMDTables[udiTableIndex].sTitle				:= 'Prepare';
	astListofCMDTables[udiTableIndex].diCMD					:= ET_Cmd.Prepare;
	astListofCMDTables[udiTableIndex].udiNumberOfCmdSteps	:= udiStepIndex;

//-------------------------------------------------------------------------------------------------------------------
//-- Auto  --
	//
	TPL.FC_FirstStep(udiStepIndex, diStep);
	astAutoTable[udiStepIndex].sTitle						:= 'Auto MultiCarrier';
	astAutoTable[udiStepIndex].udiModuleName				:= c_udiMultiCarrierTrack;
	astAutoTable[udiStepIndex].diStep						:= -diStep;
	astAutoTable[udiStepIndex].diCMD						:= 0;
	astAutoTable[udiStepIndex].timTimeOut					:= T#0MS;
	astAutoTable[udiStepIndex].xEndCMD						:= FALSE;
	
	TPL.FC_LastStep(udiStepIndex, diStep);
	astAutoTable[udiStepIndex].sTitle						:= 'End';
	astAutoTable[udiStepIndex].udiModuleName				:= 0;
	astAutoTable[udiStepIndex].diStep						:= diStep;
	astAutoTable[udiStepIndex].diCMD						:= 0;
	astAutoTable[udiStepIndex].timTimeOut					:= T#0MS;
	astAutoTable[udiStepIndex].xEndCMD						:= TRUE;
	
	TPL.FC_NextCmdTable(iq_udiTableIndex:= udiTableIndex);
	astListofCMDTables[udiTableIndex].sTitle				:= 'Auto';
	astListofCMDTables[udiTableIndex].diCMD					:= ET_Cmd.Auto;
	astListofCMDTables[udiTableIndex].udiNumberOfCmdSteps	:= udiStepIndex;

//-------------------------------------------------------------------------------------------------------------------
//-- Manual  --
	//
	TPL.FC_FirstStep(udiStepIndex, diStep);
	astManualTable[udiStepIndex].sTitle						:= 'Manual Multicarrier';
	astManualTable[udiStepIndex].udiModuleName				:= c_udiMultiCarrierTrack;
	astManualTable[udiStepIndex].diStep						:= -diStep;
	astManualTable[udiStepIndex].diCMD						:= 0;
	astManualTable[udiStepIndex].timTimeOut					:= T#0MS;
	astManualTable[udiStepIndex].xEndCMD					:= FALSE;
	
	TPL.FC_LastStep(udiStepIndex, diStep);
	astManualTable[udiStepIndex].sTitle						:= 'End';
	astManualTable[udiStepIndex].udiModuleName				:= 0;
	astManualTable[udiStepIndex].diStep						:= diStep;
	astManualTable[udiStepIndex].diCMD						:= 0;
	astManualTable[udiStepIndex].timTimeOut					:= T#0MS;
	astManualTable[udiStepIndex].xEndCMD					:= TRUE;
	
	TPL.FC_NextCmdTable(iq_udiTableIndex:= udiTableIndex);
	astListofCMDTables[udiTableIndex].sTitle				:= 'Manual';
	astListofCMDTables[udiTableIndex].diCMD					:= ET_Cmd.Manual;
	astListofCMDTables[udiTableIndex].udiNumberOfCmdSteps	:= udiStepIndex;

//-------------------------------------------------------------------------------------------------------------------
//-- TestMulticarrier --
	//
	TPL.FC_FirstStep(udiStepIndex, diStep);
	astTestMulticarrierTable[udiStepIndex].sTitle			:= 'Test Multicarrier';
	astTestMulticarrierTable[udiStepIndex].udiModuleName	:= c_udiMultiCarrierTrack;
	astTestMulticarrierTable[udiStepIndex].diStep			:= -diStep;
	astTestMulticarrierTable[udiStepIndex].diCMD			:= 0;
	astTestMulticarrierTable[udiStepIndex].timTimeOut		:= T#0MS;
	astTestMulticarrierTable[udiStepIndex].xEndCMD			:= FALSE;
	                                                        
	TPL.FC_LastStep(udiStepIndex, diStep);                  
	astTestMulticarrierTable[udiStepIndex].sTitle			:= 'End';
	astTestMulticarrierTable[udiStepIndex].udiModuleName	:= 0;
	astTestMulticarrierTable[udiStepIndex].diStep			:= diStep;
	astTestMulticarrierTable[udiStepIndex].diCMD			:= 0;
	astTestMulticarrierTable[udiStepIndex].timTimeOut		:= T#0MS;
	astTestMulticarrierTable[udiStepIndex].xEndCMD			:= TRUE;
	
	TPL.FC_NextCmdTable(iq_udiTableIndex:= udiTableIndex);
	astListofCMDTables[udiTableIndex].sTitle				:= 'Test Multicarrier';
	astListofCMDTables[udiTableIndex].diCMD					:= ET_Cmd.TestMulticarrier;
	astListofCMDTables[udiTableIndex].udiNumberOfCmdSteps	:= udiStepIndex;

//-------------------------------------------------------------------------------------------------------------------
//-- TrackCalibration --
	//
	TPL.FC_FirstStep(udiStepIndex, diStep);
	astTrackCalibrationTable[udiStepIndex].sTitle			:= 'TrackCalibration';
	astTrackCalibrationTable[udiStepIndex].udiModuleName	:= c_udiMultiCarrierTrack;
	astTrackCalibrationTable[udiStepIndex].diStep			:= -diStep;
	astTrackCalibrationTable[udiStepIndex].diCMD			:= 0;
	astTrackCalibrationTable[udiStepIndex].timTimeOut		:= T#0MS;
	astTrackCalibrationTable[udiStepIndex].xEndCMD			:= FALSE;
	                                                        
	TPL.FC_LastStep(udiStepIndex, diStep);                  
	astTrackCalibrationTable[udiStepIndex].sTitle			:= 'End';
	astTrackCalibrationTable[udiStepIndex].udiModuleName	:= 0;
	astTrackCalibrationTable[udiStepIndex].diStep			:= diStep;
	astTrackCalibrationTable[udiStepIndex].diCMD			:= 0;
	astTrackCalibrationTable[udiStepIndex].timTimeOut		:= T#0MS;
	astTestMulticarrierTable[udiStepIndex].xEndCMD			:= TRUE;
	
	TPL.FC_NextCmdTable(iq_udiTableIndex:= udiTableIndex);
	astListofCMDTables[udiTableIndex].sTitle				:= 'TrackCalibration';
	astListofCMDTables[udiTableIndex].diCMD					:= ET_Cmd.TrackCalibration;
	astListofCMDTables[udiTableIndex].udiNumberOfCmdSteps	:= udiStepIndex;
	
//-------------------------------------------------------------------------------------------------------------------
//-- Stop --
	//
	TPL.FC_FirstStep(udiStepIndex, diStep);
	astStopTable[udiStepIndex].sTitle						:= 'Stop Multicarrier';
	astStopTable[udiStepIndex].udiModuleName				:= c_udiMultiCarrierTrack;
	astStopTable[udiStepIndex].diStep						:= -diStep;
	astStopTable[udiStepIndex].diCMD						:= 0;
	astStopTable[udiStepIndex].timTimeOut					:= T#0MS;
	astStopTable[udiStepIndex].xEndCMD						:= FALSE;
	
	TPL.FC_LastStep(udiStepIndex, diStep);
	astStopTable[udiStepIndex].sTitle						:= 'End';
	astStopTable[udiStepIndex].udiModuleName				:= 0;
	astStopTable[udiStepIndex].diStep						:= diStep;
	astStopTable[udiStepIndex].diCMD						:= 0;
	astStopTable[udiStepIndex].timTimeOut					:= T#0MS;
	astStopTable[udiStepIndex].xEndCMD						:= TRUE;
	
	TPL.FC_NextCmdTable(iq_udiTableIndex:= udiTableIndex);
	astListofCMDTables[udiTableIndex].sTitle				:= 'Stop';
	astListofCMDTables[udiTableIndex].diCMD					:= ET_Cmd.Stop;
	astListofCMDTables[udiTableIndex].udiNumberOfCmdSteps	:= udiStepIndex;

//-------------------------------------------------------------------------------------------------------------------
//-- Start --
	//
	TPL.FC_FirstStep(udiStepIndex, diStep);
	astStartTable[udiStepIndex].sTitle						:= 'Start Multicarrier';
	astStartTable[udiStepIndex].udiModuleName				:= c_udiMultiCarrierTrack;
	astStartTable[udiStepIndex].diStep						:= diStep;
	astStartTable[udiStepIndex].diCMD						:= 0;
	astStartTable[udiStepIndex].timTimeOut					:= T#0MS;
	astStartTable[udiStepIndex].xEndCMD						:= FALSE;
	
	TPL.FC_LastStep(udiStepIndex, diStep);
	astStartTable[udiStepIndex].sTitle						:= 'End';
	astStartTable[udiStepIndex].udiModuleName				:= 0;
	astStartTable[udiStepIndex].diStep						:= diStep;
	astStartTable[udiStepIndex].diCMD						:= 0;
	astStartTable[udiStepIndex].timTimeOut					:= T#0MS;
	astStartTable[udiStepIndex].xEndCMD						:= TRUE;
	
	TPL.FC_NextCmdTable(iq_udiTableIndex:= udiTableIndex);
	astListofCMDTables[udiTableIndex].sTitle				:= 'Start';
	astListofCMDTables[udiTableIndex].diCMD					:= ET_Cmd.Start;
	astListofCMDTables[udiTableIndex].udiNumberOfCmdSteps	:= udiStepIndex;

//-------------------------------------------------------------------------------------------------------------------
//-- Abort --
	//
	TPL.FC_FirstStep(udiStepIndex, diStep);
	astAbortTable[udiStepIndex].sTitle						:= 'Abort Multicarrier';
	astAbortTable[udiStepIndex].udiModuleName				:= c_udiMultiCarrierTrack;
	astAbortTable[udiStepIndex].diStep						:= -diStep;
	astAbortTable[udiStepIndex].diCMD						:= 0;
	astAbortTable[udiStepIndex].timTimeOut					:= T#0MS;
	astAbortTable[udiStepIndex].xEndCMD						:= FALSE;
	
	TPL.FC_LastStep(udiStepIndex, diStep);
	astAbortTable[udiStepIndex].sTitle						:= 	'End';
	astAbortTable[udiStepIndex].udiModuleName				:= 	0;
	astAbortTable[udiStepIndex].diStep						:= 	diStep;
	astAbortTable[udiStepIndex].diCMD						:= 	0;
	astAbortTable[udiStepIndex].timTimeOut					:=	T#0MS;
	astAbortTable[udiStepIndex].xEndCMD						:= TRUE;
	
	TPL.FC_NextCmdTable(iq_udiTableIndex:= udiTableIndex);
	astListofCMDTables[udiTableIndex].sTitle				:= 'Abort';
	astListofCMDTables[udiTableIndex].diCMD					:= ET_Cmd.Abort;
	astListofCMDTables[udiTableIndex].udiNumberOfCmdSteps	:= udiStepIndex;

//-------------------------------------------------------------------------------------------------------------------
//-- Hold --
	//
	TPL.FC_FirstStep(udiStepIndex, diStep);
	astHoldTable[udiStepIndex].sTitle						:= 'Hold Multicarrier';
	astHoldTable[udiStepIndex].udiModuleName				:= c_udiMultiCarrierTrack;
	astHoldTable[udiStepIndex].diStep						:= diStep;
	astHoldTable[udiStepIndex].diCMD						:= 0;
	astHoldTable[udiStepIndex].timTimeOut					:= T#0MS;
	astHoldTable[udiStepIndex].xEndCMD						:= FALSE;
	
	TPL.FC_LastStep(udiStepIndex, diStep);
	astHoldTable[udiStepIndex].sTitle						:= 'End';
	astHoldTable[udiStepIndex].udiModuleName				:= 0;
	astHoldTable[udiStepIndex].diStep						:= diStep;
	astHoldTable[udiStepIndex].diCMD						:= 0;
	astHoldTable[udiStepIndex].timTimeOut					:= T#0MS;
	astHoldTable[udiStepIndex].xEndCMD						:= TRUE;
	
	TPL.FC_NextCmdTable(iq_udiTableIndex:= udiTableIndex);
	astListofCMDTables[udiTableIndex].sTitle				:= 'Hold';
	astListofCMDTables[udiTableIndex].diCMD					:= ET_Cmd.Hold;
	astListofCMDTables[udiTableIndex].udiNumberOfCmdSteps	:= udiStepIndex;

//
			
// End of system generated code, could be modified for your application -)
END_ACTION

ACTION Init_SubModules:
(* System generated code, could be modified for your application *)

(*** Module Group declaration ***)

aaudiSubModuleGroups[c_udiMultiCarrierGroup1-TPL.Gc_udiGroupOffset,TPL.ET_Group.Member1] := c_udiMultiCarrierTrack;				(* There is no first element of the group c_diMultiCarrierGroup1 *)
aaudiSubModuleGroups[c_udiMultiCarrierGroup1-TPL.Gc_udiGroupOffset,TPL.ET_Group.Member2] := 0;				(* There is no second element of the group c_diMultiCarrierGroup1 *)

(* End of system generated code, could be modified for your application *)


(* System generated code, do not change without consulting 'Schneider Electric Automation GmbH' - otherwise you risk instability!!!*)
xInitSubModulesException := FALSE;

//-------------------------------------------------------------------------------------------------------------------
//-- Set IDs of SubModules *)	
	//
	TPL.FC_SetSubModuleIds(	i_udiMainModuleID			:= iq_stStandardModuleItf.i_udiModuleId,
							i_pstSubModulesItf			:= ADR(astSubModuleInterface),
							i_udiNumberOfSubModules		:= c_udiNumberOfSubModules,
							q_etDiag					=> etDiag,
							q_etDiagExt					=> etDiagExtTPL);
	
	IF etDiag <> GD.ET_Diag.Ok AND NOT xInitSubModulesException THEN
		xInitSubModulesException := TRUE;
		
		stInitSubModulesException.sMsg := PDL.FC_MultiConcat(	i_sString1 := 'SetSubModuleIds - ', 
																i_sString2 := GD.FC_EtDiagToString(i_etDiag := etDiag), 
																i_sString3 := ' - ', 
																i_sString4 := TPL.FC_EtDiagExtToString(i_etDiagExt := etDiagExtTPL));
	END_IF	

//-------------------------------------------------------------------------------------------------------------------
//-- Set exception if any exception occurred *)
	//
	fbExceptionHandler.SetException(i_xExceptionActive	:= xInitSubModulesException, 
									iq_stException		:= stInitSubModulesException, 
									iq_stExceptionList	:= iq_stExceptionList);
	
	xInitSuccessful := xInitSuccessful AND NOT xInitSubModulesException;
						
	etDiag := GD.ET_Diag.Ok;
//
(* End of system generated code, do not change without consulting 'Schneider Electric Automation GmbH' - otherwise you risk instability!!!*)
END_ACTION

ACTION ControlEnable:
IF 		NOT xControlEnable 
	AND iStateControlEnable > 0 
	AND iStateControlEnable < 200 
THEN
	iStateControlEnable	:= 200;
	
ELSIF xControlEnable AND iStateControlEnable = 0 
THEN
	iStateControlEnable	:= 10;
END_IF

fbTonTimeOutControlEnable(IN := xCheckTimeOutControlEnable, PT := timTimeoutControlEnable);

CASE iStateControlEnable OF
//-------------------------------------------------------------------------------------------------------------------------------------------
//--- Enable --------------------------------------------------------------------------------------------------------------------------------
//-------------------------------------------------------------------------------------------------------------------------------------------

	//-------------------------------------------------------------------------------------------------------------------------------------------
	0: 	//--- Wait for ControlEnable = TRUE
		xCheckTimeOutControlEnable	:= FALSE;
		
	//-------------------------------------------------------------------------------------------------------------------------------------------
	10:	//--- Enable Track
		xEnableTrackSuccessful	:= FALSE;
		
		iq_stMulticarrierModule.i_ifMulticarrierTrackEnable.EnableSet := TRUE;
		xCheckTimeOutControlEnable	:= TRUE;
		
		iStateControlEnable		:= 20;
		
	//-------------------------------------------------------------------------------------------------------------------------------------------
	20: //--- Wait for Track is completly Enabled
		IF iq_stMulticarrierModule.i_ifMulticarrierTrackEnable.State = 1 THEN
			xCheckTimeOutControlEnable	:= FALSE;
			// Enable the FB_Multicarrier
			xEnableFbMulticarrier		:= TRUE;
			xStartFbMulticarrier		:= TRUE;
			iStateControlEnable			:= 30;
			
		END_IF
		
	//-------------------------------------------------------------------------------------------------------------------------------------------
	30: //--- Wait for FB_Multicarrier active 
		IF astSubModuleInterface[c_udiMultiCarrierTrack].q_xActive AND astSubModuleInterface[c_udiMultiCarrierTrack].q_xReady
		THEN
			xEnableFbCrashPrevention	:= GVL_Project.Gc_xEnableCrashPrevention;
			iStateControlEnable			:= 40;
		END_IF
		
	//-------------------------------------------------------------------------------------------------------------------------------------------
	40: //--- Check for Ready FB_Multicarrier
		IF NOT astSubModuleInterface[c_udiMultiCarrierTrack].q_xException AND astSubModuleInterface[c_udiMultiCarrierTrack].q_xReady THEN
			iStateControlEnable		:= 50;
		END_IF
		
	//-------------------------------------------------------------------------------------------------------------------------------------------
	50: //--- xEnableTrackSuccessful	
		xEnableTrackSuccessful	:= TRUE;

	
//-------------------------------------------------------------------------------------------------------------------------------------------	
//--- Disable -------------------------------------------------------------------------------------------------------------------------------
//-------------------------------------------------------------------------------------------------------------------------------------------

	//-------------------------------------------------------------------------------------------------------------------------------------------
	200:	//--- Disable FB_Multicarrier
		xEnableTrackSuccessful := FALSE;
		
		iStateControlEnable			:= 210;
		xEnableFbMulticarrier		:= FALSE;
		xStartFbMulticarrier		:= FALSE;
		xEnableFbCrashPrevention	:= FALSE;
		xEnableFbTrackCalibration	:= FALSE;
		xStartFbTrackCalibration	:= FALSE;
		
		diTimerStopOpmode			:= LMC_PacDrive.Timer1;
		
	//-------------------------------------------------------------------------------------------------------------------------------------------	
	210:	//--- Check FB_Multicarrier is disabled
		IF		NOT astSubModuleInterface[c_udiMultiCarrierTrack].q_xActive 
			AND NOT astSubModuleInterface[c_udiMultiCarrierTrack].q_xReady 
			AND NOT ifMulticarrier.ifFeedback.xMotionActiveAnyCarrier 
			AND LMC_PacDrive.Timer1 > diTimerStopOpmode + diWaitTimeSetCarrierEnableFalse
		THEN
			iStateControlEnable		:= 220;
		END_IF
		
	
	//-------------------------------------------------------------------------------------------------------------------------------------------	
	220:	//--- Disable Segments and Carrier
		iq_stMulticarrierModule.i_ifMulticarrierTrackEnable.EnableSet := FALSE;
		xCheckTimeOutControlEnable	:= TRUE;
		
		iStateControlEnable		:= 230;
		
	//-------------------------------------------------------------------------------------------------------------------------------------------
	230: //--- Check Segments and Carrier are disabled
		IF iq_stMulticarrierModule.i_ifMulticarrierTrackEnable.State = 0
		THEN	
			iStateControlEnable		:= 400;
		END_IF
	
	//-------------------------------------------------------------------------------------------------------------------------------------------
	400: //--- StopOpModeSuccessful
		IF NOT ifMulticarrier.ifFeedback.xMotionActiveAnyCarrier THEN
			xEnableFbMulticarrier		:= FALSE;
			xStartFbMulticarrier		:= FALSE;
			
			iStateControlEnable		:= 0;
		END_IF

END_CASE
END_ACTION

ACTION ControlModule:
//-- recognize error *)
fbRTrigError(CLK := xErrorActive);

//-- recognize change of OpMode or command *)
fbRTrigCMDActive(CLK := iq_stStandardModuleItf.q_xCMDActive);
	
//-- new command -> goto opmode selection state
IF fbRTrigCMDActive.Q THEN	
	ExitLastOpMode();
	iStateOpMode	:= 10;
END_IF

//-- error -> goto error state
IF fbRTrigError.Q THEN
	StoreCurrentMoveCmds();
	iStateOpMode	:= 1000;
END_IF
	
	

(*****************************************************************************************)
(*                                    Statemachine                                    	 *)
(*****************************************************************************************)

CASE iStateOpMode OF

//--------------------------------------------------------------------------------------------------------------
0:    //--- Wait
		astSubModuleInterface[c_udiMultiCarrierTrack].q_sDiagExt := 'Wait for cmd';

//-------------------------------------------------------------------------------------------------------------
10:	  //--- select Opmode 
	//
		IF (iq_stStandardModuleItf.q_diCMDActive = ET_Cmd.Auto) THEN
			etLastCmd    := ET_Cmd.Auto;
			iStateOpMode := 100;
		ELSIF (iq_stStandardModuleItf.q_diCMDActive = ET_Cmd.Prepare) THEN
			etLastCmd    := ET_Cmd.Prepare;
			iStateOpMode := 200;
		ELSIF (iq_stStandardModuleItf.q_diCMDActive = ET_Cmd.TestMulticarrier) THEN
			etLastCmd    := ET_Cmd.TestMulticarrier;
			iStateOpMode := 300;
		ELSIF (iq_stStandardModuleItf.q_diCMDActive = ET_Cmd.TrackCalibration) THEN
			etLastCmd    := ET_Cmd.TrackCalibration;
			iStateOpMode := 400;
		ELSIF (iq_stStandardModuleItf.q_diCMDActive = ET_Cmd.Manual) THEN
			etLastCmd    := ET_Cmd.Manual;
			iStateOpMode := 600;
		ELSIF (iq_stStandardModuleItf.q_diCMDActive = ET_Cmd.Stop) THEN
			etLastCmd    := ET_Cmd.Stop;
			iStateOpMode := 800;
		ELSIF (iq_stStandardModuleItf.q_diCMDActive = ET_Cmd.Abort) THEN
			etLastCmd    := ET_Cmd.Abort;
			iStateOpMode := 900;
		ELSE
			iStateOpMode := 0;
		END_IF
		
//-------------------------------------------------------------------------------------------------------------
100:  //--- OpMode Automatic
	 //--- Entry OpMode / Init  
			iq_stStandardModuleItf.iq_diStartStep := iq_stStandardModuleItf.iq_stExt.diActiveStep + 10;
			iStateOpMode := 110;
			
	110:	//--- Automatic active
			IF 		NOT iq_stStandardModuleItf.q_xCMDActive
				AND iq_stStandardModuleItf.q_xCmdDone
				AND astSubModuleInterface[c_udiMultiCarrierTrack].q_xActive
			THEN
				astSubModuleInterface[c_udiMultiCarrierTrack].q_sDiagExt := 'Multicarrier Running';
				uiSetOpModeVis 				:= ET_OpModeVis.Auto;
				xSetStationTriggerViaTimer	:= FALSE;
				xStartFbCrashPrevention		:= TRUE;
				iStateOpMode 				:= 120;
			END_IF
			
	120:	//--- cyclic call  
			CallAllStations();

//-------------------------------------------------------------------------------------------------------------
200:  //--- OpMode Prepare
	 //---  Entry OpMode / Init  
		xHomingWasSuccessful	:= FALSE; 
		xControlEnable			:= TRUE; 
		
		astSubModuleInterface[c_udiMultiCarrierTrack].q_sDiagExt := 'Prepare running';
		iStateOpMode := 210;
			
	210:	//--- call parameter of station1
			IF 		xWaitForStartStep
				AND	xEnableTrackSuccessful 
				AND NOT astSubModuleInterface[c_udiMultiCarrierTrack].q_xCmdActive 
			THEN
				iStateOpMode := 220;
			END_IF
				
	220:	//--- Wait until FB_Multicarrier is Ready 
			IF 		astSubModuleInterface[c_udiMultiCarrierTrack].q_xActive 
				AND	astSubModuleInterface[c_udiMultiCarrierTrack].q_xReady
				AND	etResultFbMulticarrier = MCR.ET_Result.Working
			THEN
				IF GVL_Project.Gc_xVirtualMulticarrier AND iq_stMulticarrierModule.iq_xDoVirtualSetposAfterFirstProgramCall THEN	
					iStateOpMode := 230;
				ELSE
					iStateOpMode := 240;
				END_IF		
			END_IF
			
	230:	//--- in case of virtual multicarrer -> setpos on all carriers
			IF VirtualSetPosOfAllCarriers() THEN
				iq_stMulticarrierModule.iq_xDoVirtualSetposAfterFirstProgramCall := FALSE;
				iStateOpMode := 240;
			END_IF
			
	240:	//--- move carriers in first station
			DeleteAllCarriersFromStations();
			ParameterStation1();
			MoveAllCarriersInFirstStation();
			IF NOT xSetException THEN
				iStateOpMode := 250;
			END_IF
			
			
	250:	//--- Reset wait step of cmd-table
			IF 		xWaitForStartStep 
				AND	NOT ifMulticarrier.ifFeedback.xMotionActiveAnyCarrier
			THEN
				iq_stStandardModuleItf.iq_diStartStep := iq_stStandardModuleItf.iq_stExt.diActiveStep + 10;
				iStateOpMode := 260;
			END_IF
				
	260:	//--- End cmd table 
			IF 		NOT iq_stStandardModuleItf.q_xCMDActive
				AND	iq_stStandardModuleItf.q_xCmdDone 
			THEN	
				astSubModuleInterface[c_udiMultiCarrierTrack].q_sDiagExt := 'Prepare done';
				xHomingWasSuccessful	:= TRUE; 
				iStateOpMode	:= 0;			
			END_IF


//-------------------------------------------------------------------------------------------------------------
300:  //--- OpMode TestMulticarrier
	 //---  Entry OpMode / Init  
			xControlEnable			:= TRUE; 
			xHomingWasSuccessful	:= FALSE; 
			iStateOpMode 			:= 310;

	310:	//--- Wait until FB_Multicarrier is Ready 
			IF 		astSubModuleInterface[c_udiMultiCarrierTrack].q_xActive 
				AND	astSubModuleInterface[c_udiMultiCarrierTrack].q_xReady
				AND	etResultFbMulticarrier = MCR.ET_Result.Working
			THEN
				uiSetOpModeVis 	:= ET_OpModeVis.Test;
				DeleteAllCarriersFromStations();
				iStateOpMode 	:= 320;
			END_IF
			
	320:	//--- check for virtual setpos
			IF GVL_Project.Gc_xVirtualMulticarrier  AND_THEN iq_stMulticarrierModule.iq_xDoVirtualSetposAfterFirstProgramCall THEN	
				iStateOpMode := 330;
			ELSE
				iStateOpMode := 340;
				StopAllCarriers();
			END_IF		
			
	330:	//--- in case of virtual multicarrer -> setpos on all carriers
			IF VirtualSetPosOfAllCarriers() THEN
				iq_stMulticarrierModule.iq_xDoVirtualSetposAfterFirstProgramCall := FALSE;
				iStateOpMode := 340;
			END_IF
			
	340:	IF	xWaitForStartStep THEN
				astSubModuleInterface[c_udiMultiCarrierTrack].q_sDiagExt := 'Test Multicarrier Running';
				//--- reset wait step of cmd-table
				iq_stStandardModuleItf.iq_diStartStep := iq_stStandardModuleItf.iq_stExt.diActiveStep + 10;
				
				iStateOpMode := 350;
			END_IF
			
	350:	//--- cyclic call of test stations 
			SR_CallTestStations(
					i_etTraceSource		:= etTraceSource,
					i_ifMultiCarrier	:= fbMulticarrier,
					i_xStart			:= xStartTest,
					i_xStop				:= xStopTest,
					q_xError			=> xSetException,
					q_sEtResult			=> stException.sDiagExt,
					q_sResultMsg		=> sResultMsgMCR);	
					
//-------------------------------------------------------------------------------------------------------------
400:  //--- OpMode TrackCalibration
	 //---  Entry OpMode / Init  
			xControlEnable			:= TRUE; 
			xHomingWasSuccessful	:= FALSE; 
			iStateOpMode 			:= 410;

	410:	//--- Wait until FB_Multicarrier is Ready 
			IF 		astSubModuleInterface[c_udiMultiCarrierTrack].q_xActive 
				AND	astSubModuleInterface[c_udiMultiCarrierTrack].q_xReady
				AND	etResultFbMulticarrier = MCR.ET_Result.Working
			THEN
				uiSetOpModeVis 	:= ET_OpModeVis.TrackCalibration;
				DeleteAllCarriersFromStations();
				iStateOpMode 	:= 420;
			END_IF
			
	420:	//--- Enable FB_TrackCalibration
			StopAllCarriers();
			xEnableFbTrackCalibration 	:= TRUE;
			xStartFbTrackCalibration	:= TRUE;
			iStateOpMode := 430;
			
	430:	//--- Check if FB_TrackCalibration is active and ready
			IF xActiveFbTrackCalibration
			AND xReadyFbTrackCalibration
			THEN
				iStateOpMode := 440;
			END_IF
			
	440:	IF	xWaitForStartStep THEN
				astSubModuleInterface[c_udiMultiCarrierTrack].q_sDiagExt := 'TrackCalibration';
				//--- reset wait step of cmd-table
				iq_stStandardModuleItf.iq_diStartStep := iq_stStandardModuleItf.iq_stExt.diActiveStep + 10;
				
				iStateOpMode := 450;
			END_IF
			
	450:	//--- cyclic call of SR_CallTrackCalibration
			TrackCalibration_Logic();
			
//-------------------------------------------------------------------------------------------------------------
600:  //--- OpMode Manual 
	 //---  Entry OpMode / Init  
			xControlEnable			:= TRUE; 
			xHomingWasSuccessful	:= FALSE; 
			iStateOpMode 			:= 610;
			
	610:	//--- wait for FB_Multicarrier is ready
			IF 		xWaitForStartStep 	
				AND	astSubModuleInterface[c_udiMultiCarrierTrack].q_xActive 
				AND	astSubModuleInterface[c_udiMultiCarrierTrack].q_xReady
				AND	etResultFbMulticarrier = MCR.ET_Result.Working
			THEN
				IF GVL_Project.Gc_xVirtualMulticarrier AND_THEN iq_stMulticarrierModule.iq_xDoVirtualSetposAfterFirstProgramCall THEN	
					iStateOpMode := 620;
				ELSE
					//--- reset wait step of cmd-table
					iq_stStandardModuleItf.iq_diStartStep := iq_stStandardModuleItf.iq_stExt.diActiveStep + 10;	
					iStateOpMode := 630;
				END_IF		
			END_IF
			
	620:	//--- in case of virtual multicarrer -> setpos on all carriers
			IF VirtualSetPosOfAllCarriers() THEN
				iq_stMulticarrierModule.iq_xDoVirtualSetposAfterFirstProgramCall := FALSE;
				//--- reset wait step of cmd-table
				iq_stStandardModuleItf.iq_diStartStep := iq_stStandardModuleItf.iq_stExt.diActiveStep + 10;	
				iStateOpMode := 630;
			END_IF
			
	630:	//--- Manual is active
			IF 		NOT iq_stStandardModuleItf.q_xCMDActive
				AND	iq_stStandardModuleItf.q_xCmdDone 
			THEN	
				//--- initialize manual mode	
				uiSetOpModeVis := ET_OpModeVis.Manual;
				astSubModuleInterface[c_udiMultiCarrierTrack].q_sDiagExt := 'Manual running';
				Manual_Entry();
				iStateOpMode	:= 640;
			END_IF
			
	640:	//--- cyclic call
			Manual_Logic();

//-------------------------------------------------------------------------------------------------------------
800:  //--- OpMode Stop 
	//
			IF 		astSubModuleInterface[c_udiMultiCarrierTrack].q_xActive 
				AND	astSubModuleInterface[c_udiMultiCarrierTrack].q_xReady
				AND	etResultFbMulticarrier = MCR.ET_Result.Working
			THEN
				SR_CallTestStations.ResetStateAndTrigger();
				StopAllCarriers();
				iStateOpMode	:= 810;	
			ELSE
				//--- reset wait step of cmd-table
				iq_stStandardModuleItf.iq_diStartStep := iq_stStandardModuleItf.iq_stExt.diActiveStep + 10;
				iStateOpMode	:= 820;	
			END_IF
			
	810:	IF NOT ifMulticarrier.ifFeedback.xMotionActiveAnyCarrier THEN
				xStartFbCrashPrevention	:= FALSE;
				xEnableFbTrackCalibration	:= FALSE;
				xStartFbTrackCalibration	:= FALSE;
				
				//--- reset wait step of cmd-table
				iq_stStandardModuleItf.iq_diStartStep := iq_stStandardModuleItf.iq_stExt.diActiveStep + 10;
				iStateOpMode	:= 820;	
			END_IF
			
			
 	820:	//--- End cmd table 
			IF 		NOT iq_stStandardModuleItf.q_xCMDActive
				AND	iq_stStandardModuleItf.q_xCmdDone 
			THEN	
				xHomingWasSuccessful	:= FALSE; 
				astSubModuleInterface[c_udiMultiCarrierTrack].q_sDiagExt := 'Stop done';
				uiSetOpModeVis 	:= ET_OpModeVis.None;
				iStateOpMode	:= 0;			
			END_IF
			
//-------------------------------------------------------------------------------------------------------------
900:  //--- OpMode Abort 
	//
			IF 		astSubModuleInterface[c_udiMultiCarrierTrack].q_xActive 
				AND	astSubModuleInterface[c_udiMultiCarrierTrack].q_xReady
				AND	etResultFbMulticarrier = MCR.ET_Result.Working
			THEN
				SR_CallTestStations.ResetStateAndTrigger();
				StopAllCarriers();
				iStateOpMode	:= 910;	
			ELSE
				//--- reset wait step of cmd-table
				iq_stStandardModuleItf.iq_diStartStep := iq_stStandardModuleItf.iq_stExt.diActiveStep + 10;
				iStateOpMode	:= 920;	
			END_IF
			
	910:	IF NOT ifMulticarrier.ifFeedback.xMotionActiveAnyCarrier THEN
				xStartFbCrashPrevention	:= FALSE;
				//--- reset wait step of cmd-table
				iq_stStandardModuleItf.iq_diStartStep := iq_stStandardModuleItf.iq_stExt.diActiveStep + 10;
				iStateOpMode	:= 920;	
			END_IF
			
			
 	920:	//--- End cmd table 
			IF 		NOT iq_stStandardModuleItf.q_xCMDActive
				AND	iq_stStandardModuleItf.q_xCmdDone 
			THEN	
				xHomingWasSuccessful	:= FALSE; 
				astSubModuleInterface[c_udiMultiCarrierTrack].q_sDiagExt := 'Abort done';
				uiSetOpModeVis 	:= ET_OpModeVis.None;
				iStateOpMode	:= 0;			
			END_IF
			
//-------------------------------------------------------------------------------------------------------------
1000: //--- Command Error 
	//
			//-- reset homing signal
			xHomingWasSuccessful			:= FALSE; 
			//-- stop all Carriers and disable track in Action ControlEnable 
			xControlEnable					:= FALSE;
			
			//-- reset vis
	 		uiSetOpModeVis 	:= ET_OpModeVis.None;
			iStateOpMode	:= 1010;
			
	1010:	//--  Wait for acknowledge of the fault 
			IF iq_stStandardModuleItf.i_xDiagQuit THEN
				//--  Reset Error 
				ErrorQuitStations();				
				xSetException				:= FALSE;
				xErrorStored				:= FALSE;
				
				stException.udiDiagExt		:= 0;
				stException.sDiagExt		:= '';
				stException.sMsg			:= '';
				sResultMsgMCR				:= '';
				sResultMsg1					:= '';
				sResultMsg2					:= '';
				sResultMsg3					:= '';
				
				SR_CallTestStations.ErrorQuit();
				iStateOpMode	:= 0;
			END_IF
//-------------------------------------------------------------------------------------------------------------

END_CASE
END_ACTION

METHOD AddMessageToAPL : BOOL
VAR_INPUT
	i_sMsg : STRING(255);
END_VAR

VAR_STAT
	sMsgOld : STRING(255);
END_VAR
IF i_sMsg <> sMsgOld THEN	
	
	sMsgOld := i_sMsg;
	
	fbLoggerPoint.AddLogEntry(	i_etLogLevel	:= APL.ET_LogLevel.UserAction,
								i_etDiag		:= 0,
								i_udiDiagExt	:= APL.ET_DiagExt.Ok,
								i_sMessage		:= i_sMsg,
								q_etDiag		=> ,
								q_etDiagExt		=> );
END_IF
END_METHOD

METHOD APLStartPosEndPos
VAR_INPUT
	i_lrStartPos 	: LREAL;
	i_lrEndPos		: LREAL;
END_VAR

VAR
	udiCarrierIndex		: UDINT;
END_VAR
//--- add carrier to aplicationlogger
		FOR udiCarrierIndex := 1 TO fbMulticarrier.ifFeedback.ifFeedbackConfiguration.udiNumberOfCarriers DO
			//--- Check if Carrier is inside start and end pos
				//--- zero is not inside start and end pos 
				IF i_lrStartPos < i_lrEndPos THEN 
					IF 		fbMulticarrier.raifCarrier[udiCarrierIndex].ifFeedback.ifFeedbackMotionValues.lrRefTrackPosition >= i_lrStartPos
						AND fbMulticarrier.raifCarrier[udiCarrierIndex].ifFeedback.ifFeedbackMotionValues.lrRefTrackPosition <= i_lrEndPos
						AND NOT fbMulticarrier.raifCarrier[udiCarrierIndex].ifFeedback.ifFeedbackConfiguration.xApplicationLoggerEntriesActive
					THEN
						fbMulticarrier.raifCarrier[udiCarrierIndex].ifConfiguration.ConfigureApplicationLoggerEntries(i_xApplicationLoggerEntriesActive := TRUE);
					END_IF
					
				//--- zero is inside start and end pos  
				ELSIF i_lrStartPos > i_lrEndPos THEN 
					IF 		(fbMulticarrier.raifCarrier[udiCarrierIndex].ifFeedback.ifFeedbackMotionValues.lrRefTrackPosition >= i_lrStartPos
							  OR fbMulticarrier.raifCarrier[udiCarrierIndex].ifFeedback.ifFeedbackMotionValues.lrRefTrackPosition <= i_lrEndPos
							)
						AND NOT fbMulticarrier.raifCarrier[udiCarrierIndex].ifFeedback.ifFeedbackConfiguration.xApplicationLoggerEntriesActive
					THEN
						fbMulticarrier.raifCarrier[udiCarrierIndex].ifConfiguration.ConfigureApplicationLoggerEntries(i_xApplicationLoggerEntriesActive := TRUE);
					END_IF
				END_IF
		END_FOR
		
	//--- delete carrier to aplicationlogger
		FOR udiCarrierIndex := 1 TO fbMulticarrier.ifFeedback.ifFeedbackConfiguration.udiNumberOfCarriers DO
			//--- Check if Carrier is outside
				//--- zero is not inside start and end pos 
				IF i_lrStartPos < i_lrEndPos THEN 
					IF 		(fbMulticarrier.raifCarrier[udiCarrierIndex].ifFeedback.ifFeedbackMotionValues.lrRefTrackPosition >= i_lrEndPos
							  OR fbMulticarrier.raifCarrier[udiCarrierIndex].ifFeedback.ifFeedbackMotionValues.lrRefTrackPosition <= i_lrStartPos
							)
						AND fbMulticarrier.raifCarrier[udiCarrierIndex].ifFeedback.ifFeedbackConfiguration.xApplicationLoggerEntriesActive
					THEN
						fbMulticarrier.raifCarrier[udiCarrierIndex].ifConfiguration.ConfigureApplicationLoggerEntries(i_xApplicationLoggerEntriesActive := FALSE);
					END_IF
					
				//--- zero is inside start and end pos  
				ELSIF i_lrStartPos > i_lrEndPos THEN 
					IF 		fbMulticarrier.raifCarrier[udiCarrierIndex].ifFeedback.ifFeedbackMotionValues.lrRefTrackPosition >= i_lrEndPos
						AND fbMulticarrier.raifCarrier[udiCarrierIndex].ifFeedback.ifFeedbackMotionValues.lrRefTrackPosition <= i_lrStartPos
						AND fbMulticarrier.raifCarrier[udiCarrierIndex].ifFeedback.ifFeedbackConfiguration.xApplicationLoggerEntriesActive
					THEN
						fbMulticarrier.raifCarrier[udiCarrierIndex].ifConfiguration.ConfigureApplicationLoggerEntries(i_xApplicationLoggerEntriesActive := FALSE);
					END_IF
				END_IF
		END_FOR
END_METHOD

ACTION TraceAndAPL:
//-------------------------------------------------------------------------------------------------------------------------------------------
//--- Set Traceobjects
//-------------------------------------------------------------------------------------------------------------------------------------------
	IF etTraceSource = ET_TraceSource.MulticarrierModule OR etTraceSource = ET_TraceSource.StartPosAndEndPos THEN
		
		IF etTraceSource = ET_TraceSource.StartPosAndEndPos THEN
			TraceStartPosEndPos(i_lrStartPos:= lrTraceStartTrackPos, i_lrEndPos:= lrTraceEndTrackPos);
		END_IF
		
		aifTraceObject[1] := fbMulticarrier.raifCarrier[LIMIT(1,udiTraceObject1,ifMulticarrier.ifFeedback.ifFeedbackConfiguration.udiNumberOfCarriers)].ifFeedback;
		aifTraceObject[2] := fbMulticarrier.raifCarrier[LIMIT(1,udiTraceObject2,ifMulticarrier.ifFeedback.ifFeedbackConfiguration.udiNumberOfCarriers)].ifFeedback;
		aifTraceObject[3] := fbMulticarrier.raifCarrier[LIMIT(1,udiTraceObject3,ifMulticarrier.ifFeedback.ifFeedbackConfiguration.udiNumberOfCarriers)].ifFeedback;
		aifTraceObject[4] := fbMulticarrier.raifCarrier[LIMIT(1,udiTraceObject4,ifMulticarrier.ifFeedback.ifFeedbackConfiguration.udiNumberOfCarriers)].ifFeedback;
		aifTraceObject[5] := fbMulticarrier.raifCarrier[LIMIT(1,udiTraceObject5,ifMulticarrier.ifFeedback.ifFeedbackConfiguration.udiNumberOfCarriers)].ifFeedback;
		
		aifTraceCarrierMovementData[1] := iq_stMulticarrierModule.i_aifMovementData[LIMIT(1,udiTraceObject1,ifMulticarrier.ifFeedback.ifFeedbackConfiguration.udiNumberOfCarriers)];
		aifTraceCarrierMovementData[2] := iq_stMulticarrierModule.i_aifMovementData[LIMIT(1,udiTraceObject2,ifMulticarrier.ifFeedback.ifFeedbackConfiguration.udiNumberOfCarriers)];
		aifTraceCarrierMovementData[3] := iq_stMulticarrierModule.i_aifMovementData[LIMIT(1,udiTraceObject3,ifMulticarrier.ifFeedback.ifFeedbackConfiguration.udiNumberOfCarriers)];
		aifTraceCarrierMovementData[4] := iq_stMulticarrierModule.i_aifMovementData[LIMIT(1,udiTraceObject4,ifMulticarrier.ifFeedback.ifFeedbackConfiguration.udiNumberOfCarriers)];
		aifTraceCarrierMovementData[5] := iq_stMulticarrierModule.i_aifMovementData[LIMIT(1,udiTraceObject5,ifMulticarrier.ifFeedback.ifFeedbackConfiguration.udiNumberOfCarriers)];
		
	ELSE
		
		SR_CarriersInStationToTrace(
				i_xOneByOne					:= xOneByOne,
				i_udiNumberOfCarrierInTrace := udiNumberOfCarrierInTrace,
				i_ifMultiCarrier  			:= fbMulticarrier,
				iq_xReStartSerialCount 		:= xReStartOneByOneCount,
				q_aifTraceObject  			=> aifTraceObject);
				
	END_IF

//-------------------------------------------------------------------------------------------------------------------------------------------
//--- ApplicationLogger
//-------------------------------------------------------------------------------------------------------------------------------------------
	IF etLogLevelMcr <> etLogLevelMcrOld THEN
		etLogLevelMcrOld	:= etLogLevelMcr;
		ifMulticarrier.SetApplicationLoggerLogLevel(i_etLogLevel := etLogLevelMcr);
		fbTrackCalibration.SetApplicationLoggerLogLevel(i_etLogLevel := etLogLevelMcr);
	END_IF
	
	IF xSetForAllAplMsg THEN
		xSetForAllAplMsg := FALSE;
		FOR udiLoop := 1 TO ifMulticarrier.ifFeedback.ifFeedbackConfiguration.udiNumberOfCarriers DO
			ifMulticarrier.raifCarrier[udiLoop].ifConfiguration.ConfigureApplicationLoggerEntries(i_xApplicationLoggerEntriesActive := TRUE);
		END_FOR
	END_IF
	
	IF xReSetForAllAplMsg THEN
		xReSetForAllAplMsg := FALSE;
		FOR udiLoop := 1 TO ifMulticarrier.ifFeedback.ifFeedbackConfiguration.udiNumberOfCarriers DO
			ifMulticarrier.raifCarrier[udiLoop].ifConfiguration.ConfigureApplicationLoggerEntries(i_xApplicationLoggerEntriesActive := FALSE);
		END_FOR
	END_IF
	
	IF xSetSingleAplMsg THEN
		xSetSingleAplMsg := FALSE;
		IF ifMulticarrier.raifCarrier[udiSingleCarrierNr].ifFeedback.ifFeedbackConfiguration.xApplicationLoggerEntriesActive THEN
			ifMulticarrier.raifCarrier[udiSingleCarrierNr].ifConfiguration.ConfigureApplicationLoggerEntries(i_xApplicationLoggerEntriesActive := FALSE);
		ELSE
			ifMulticarrier.raifCarrier[udiSingleCarrierNr].ifConfiguration.ConfigureApplicationLoggerEntries(i_xApplicationLoggerEntriesActive := TRUE);
		END_IF
	END_IF
		
	IF xAplMsgStartPosAndEndPos THEN
		APLStartPosEndPos(i_lrStartPos:= lrAplStartTrackPos, i_lrEndPos:= lrAplEndTrackPos);
	END_IF

	//--- calculation for Vis
	IF udiDeltaBottomY = 1000 THEN
	 	udiDeltaBottomY := ((ifMulticarrier.ifFeedback.ifFeedbackConfiguration.udiNumberOfCarriers - 1) / 10) * 40;
	END_IF
	IF etTraceSource = ET_TraceSource.StartPosAndEndPos THEN
		iTopTraceEntryVis := 0;
	ELSE
		iTopTraceEntryVis := -55;
	END_IF

//
END_ACTION

METHOD TraceStartPosEndPos

VAR CONSTANT
	c_udiTraceObjects : UDINT := 5;
END_VAR

VAR_INPUT
	i_lrStartPos 	: LREAL;
	i_lrEndPos		: LREAL;
END_VAR

VAR_STAT
	udiNbOfCarrier 			: UDINT;
	axCarrierArrayIsBlocked : ARRAY [1..c_udiTraceObjects] OF BOOL;
	audiTraceCarrierIndex 	: ARRAY [1..c_udiTraceObjects] OF UDINT;
	udiStartIndex			: UDINT := 1;
	udiNewStartIndex		: UDINT := 1;
	udiEndIndex				: UDINT;
END_VAR

VAR
	udiCarrierIndex		: UDINT;
	udiTraceArrayIndex	: UDINT;
	xCarrierIsInside	: BOOL;
	xCarrierIsOutside	: BOOL;
	xContinue			: BOOL;
END_VAR
//--- add carrier to trace
		IF udiNbOfCarrier < c_udiTraceObjects THEN
			
			udiStartIndex	:= udiNewStartIndex;
			udiEndIndex 	:= udiStartIndex - 1;
				
			FOR udiCarrierIndex := udiStartIndex TO fbMulticarrier.ifFeedback.ifFeedbackConfiguration.udiNumberOfCarriers DO
				IF udiNbOfCarrier >= c_udiTraceObjects THEN
					EXIT;
				END_IF
				//--- Check if carrier is already added	
				FOR udiTraceArrayIndex := 1 TO c_udiTraceObjects DO
					IF audiTraceCarrierIndex[udiTraceArrayIndex] = 0 THEN
						CONTINUE;
					END_IF
					IF aifTraceObject[udiTraceArrayIndex].udiCarrierIndex = udiCarrierIndex THEN
						xContinue := TRUE;
						EXIT;
					END_IF
				END_FOR
				IF xContinue THEN
					xContinue := FALSE;
					CONTINUE;
				END_IF
				//--- Check if Carrier is inside start and end pos
					//--- zero is not inside start and end pos 
					IF i_lrStartPos < i_lrEndPos THEN 
						IF fbMulticarrier.raifCarrier[udiCarrierIndex].ifFeedback.ifFeedbackMotionValues.lrRefTrackPosition >= i_lrStartPos
							AND fbMulticarrier.raifCarrier[udiCarrierIndex].ifFeedback.ifFeedbackMotionValues.lrRefTrackPosition <= i_lrEndPos
						THEN
							xCarrierIsInside := TRUE;
						END_IF
						
					//--- zero is inside start and end pos  
					ELSIF i_lrStartPos > i_lrEndPos THEN 
						IF fbMulticarrier.raifCarrier[udiCarrierIndex].ifFeedback.ifFeedbackMotionValues.lrRefTrackPosition >= i_lrStartPos
							OR fbMulticarrier.raifCarrier[udiCarrierIndex].ifFeedback.ifFeedbackMotionValues.lrRefTrackPosition <= i_lrEndPos
						THEN
							xCarrierIsInside := TRUE;
						END_IF
					END_IF
				
				IF xCarrierIsInside	THEN
					xCarrierIsInside := FALSE;
					udiNbOfCarrier := udiNbOfCarrier + 1;
					FOR udiTraceArrayIndex := 1 TO c_udiTraceObjects DO
						IF NOT axCarrierArrayIsBlocked[udiTraceArrayIndex] THEN
							axCarrierArrayIsBlocked[udiTraceArrayIndex] := TRUE;
							audiTraceCarrierIndex[udiTraceArrayIndex] := udiCarrierIndex;
							IF udiTraceArrayIndex = 1 THEN
								udiTraceObject1	:= udiCarrierIndex;
							ELSIF udiTraceArrayIndex = 2 THEN
								udiTraceObject2	:= udiCarrierIndex;
							ELSIF udiTraceArrayIndex = 3 THEN
								udiTraceObject3	:= udiCarrierIndex;
							ELSIF udiTraceArrayIndex = 4 THEN
								udiTraceObject4	:= udiCarrierIndex;
							ELSIF udiTraceArrayIndex = 5 THEN
								udiTraceObject5	:= udiCarrierIndex;
							END_IF
							udiNewStartIndex := udiCarrierIndex;	
							EXIT;
						END_IF
					END_FOR
					
				END_IF
			END_FOR
				
			FOR udiCarrierIndex := 1 TO udiEndIndex DO
				IF udiNbOfCarrier >= c_udiTraceObjects THEN
					EXIT;
				END_IF
				//--- Check if carrier is already added	
				FOR udiTraceArrayIndex := 1 TO c_udiTraceObjects DO
					IF audiTraceCarrierIndex[udiTraceArrayIndex] = 0 THEN
						CONTINUE;
					END_IF
					IF aifTraceObject[udiTraceArrayIndex].udiCarrierIndex = udiCarrierIndex THEN
						xContinue := TRUE;
						EXIT;
					END_IF
				END_FOR
				IF xContinue THEN
					xContinue := FALSE;
					CONTINUE;
				END_IF
				//--- Check if Carrier is inside start and end pos
					//--- zero is not inside start and end pos 
					IF i_lrStartPos < i_lrEndPos THEN 
						IF fbMulticarrier.raifCarrier[udiCarrierIndex].ifFeedback.ifFeedbackMotionValues.lrRefTrackPosition >= i_lrStartPos
							AND fbMulticarrier.raifCarrier[udiCarrierIndex].ifFeedback.ifFeedbackMotionValues.lrRefTrackPosition <= i_lrEndPos
						THEN
							xCarrierIsInside := TRUE;
						END_IF
						
					//--- zero is inside start and end pos  
					ELSIF i_lrStartPos > i_lrEndPos THEN 
						IF fbMulticarrier.raifCarrier[udiCarrierIndex].ifFeedback.ifFeedbackMotionValues.lrRefTrackPosition >= i_lrStartPos
							OR fbMulticarrier.raifCarrier[udiCarrierIndex].ifFeedback.ifFeedbackMotionValues.lrRefTrackPosition <= i_lrEndPos
						THEN
							xCarrierIsInside := TRUE;
						END_IF
					END_IF
				
				IF xCarrierIsInside	THEN
					xCarrierIsInside := FALSE;
					udiNbOfCarrier := udiNbOfCarrier + 1;
					FOR udiTraceArrayIndex := 1 TO c_udiTraceObjects DO
						IF NOT axCarrierArrayIsBlocked[udiTraceArrayIndex] THEN
							axCarrierArrayIsBlocked[udiTraceArrayIndex] := TRUE;
							audiTraceCarrierIndex[udiTraceArrayIndex] := udiCarrierIndex;
							IF udiTraceArrayIndex = 1 THEN
								udiTraceObject1	:= udiCarrierIndex;
							ELSIF udiTraceArrayIndex = 2 THEN
								udiTraceObject2	:= udiCarrierIndex;
							ELSIF udiTraceArrayIndex = 3 THEN
								udiTraceObject3	:= udiCarrierIndex;
							ELSIF udiTraceArrayIndex = 4 THEN
								udiTraceObject4	:= udiCarrierIndex;
							ELSIF udiTraceArrayIndex = 5 THEN
								udiTraceObject5	:= udiCarrierIndex;
							END_IF	
							udiNewStartIndex := udiCarrierIndex;	
							EXIT;
						END_IF
					END_FOR
				END_IF
			END_FOR

		END_IF
		
